       "DB_McpKeyboardSignals".sK5_GripperDrilledPart.sLedSWStatus := "DB_McpKeyboardSignals".sK5_GripperDrilledPart.sKeySWStatus;
       "DB_HmiKeyboardSignals".sK5a_GripperDrilledPartClose.sLedSWStatus := "DB_HmiKeyboardSignals".sK5a_GripperDrilledPartClose.sKeySWStatus;
       "DB_HmiKeyboardSignals".sK5b_GripperDrilledPartOpen.sLedSWStatus := "DB_HmiKeyboardSignals".sK5b_GripperDrilledPartOpen.sKeySWStatus;
   END_REGION

   REGION Undrilled Gripper        
       #sUndrilledGripper(iHoldPart := #sLoadGripperCloseReq,
                          iOpen := "DB_DigitalInputs".sLoadClampOpened.sSWStatus,
                          iCloseWithoutPart := "DB_DigitalInputs".sLoadClampNotClosedWithPart.sSWStatus,
                          iPulseTime := T#300ms,
                          iMonitorTime:=T#3s,
                          oClose => "DB_DigitalOutputs".sLoadClampClosing.sSWStatus,
                          oOpen => "DB_DigitalOutputs".sLoadClampOpening.sSWStatus,
                          oStateOpen => #sLoadOpen,
                          oStateClose => #sLoadClose,
                          oStateCloseWithPart => #sLoadCloseWithPart,
                          oErrorCode=>#sUndrilledGripperErrorCode);

       "LBP_AlarmMsgs".UserA[08].A70UUxx[14] := #sUndrilledGripperErrorCode = 1;    // Msg: 700814 "Loading Gripper Opening Timeout"
       "LBP_AlarmMsgs".UserA[08].A70UUxx[15] := #sUndrilledGripperErrorCode = 2;    // Msg: 700815 "Loading Gripper Closing Timeout"   
   END_REGION

   REGION Drilled Gripper
       #sDrilledGripper(iHoldPart := #sUnloadGripperCloseReq,
                        iOpen := "DB_DigitalInputs".sUnloadClampOpened.sSWStatus,
                        iCloseWithoutPart := "DB_DigitalInputs".sUnloadClampNotClosedWithPart.sSWStatus,
                        iPulseTime := T#300ms,
                        iMonitorTime:=T#3s,
                        oClose => "DB_DigitalOutputs".sUnloadClampClosing.sSWStatus,
                        oOpen => "DB_DigitalOutputs".sUnloadClampOpening.sSWStatus,
                        oStateOpen => #sUnLoadOpen,
                        oStateClose => #sUnLoadClose,
                        oStateCloseWithPart => #sUnLoadCloseWithPart,
                        oErrorCode=>#sDrilledGripperErrorCode);

       "LBP_AlarmMsgs".UserA[08].A70UUxx[16] := #sUndrilledGripperErrorCode = 1;    // Msg: 700816 "Unloading Gripper Opening Timeout"
       "LBP_AlarmMsgs".UserA[08].A70UUxx[17] := #sUndrilledGripperErrorCode = 2;    // Msg: 700817 "Unloading Gripper Closing Timeout"   
   END_REGION

   REGION Blowing
       // Blowing from ISO Code
       IF "LBP_Chan1".MDyn[96] THEN
           #sBlowingISO := TRUE;
       ELSIF "LBP_Chan1".MDyn[97] OR "LBP_Chan1".A_Reset THEN
           #sBlowingISO := FALSE;
       END_IF;

       #sRT_BlowingCmdHMI(CLK := "DB_HMICmd".BlowingCmd);

       #sBlowingTimerCmdHMI(IN := #sRT_BlowingCmdHMI.Q,
                      PT := REAL_TO_DINT("DB_HMISetting".BlowingSetpoint));

       "DB_DigitalOutputs".sBlowing.sSWStatus := "DB_LoaderShuttle1".oBlowingReq
       OR "DB_LoaderShuttle2".oBlowingReq
       OR "DB_LoaderFixture".oBlowingReq
       OR  #sBlowingTimerCmdHMI.Q;

       "DB_HMICmd".BlowingCmd := FALSE;
   END_REGION

   REGION Gripper Status
       IF "DB_LoaderShuttle1".sMain.oGripperAxisRequest AND #sGripperStatus.Available AND NOT "DB_CommPLC_ISO".sAxisReservedbyNC THEN
           #sGripperStatus.Available := FALSE;
           #sGripperStatus.DrivedByShuttle1 := TRUE;
           #sGripperStatus.DrivedByShuttle2 := FALSE;
           #sGripperStatus.DrivedByFixture := FALSE;
       ELSIF "DB_LoaderShuttle2".sMain.oGripperAxisRequest AND #sGripperStatus.Available  AND NOT "DB_CommPLC_ISO".sAxisReservedbyNC THEN
           #sGripperStatus.Available := FALSE;
           #sGripperStatus.DrivedByShuttle1 := FALSE;
           #sGripperStatus.DrivedByShuttle2 := TRUE;
           #sGripperStatus.DrivedByFixture := FALSE;
       ELSIF #sGripperReq.ByFixture AND #sGripperStatus.Available  AND "DB_CommPLC_ISO".sAxisReservedbyNC THEN
           #sGripperStatus.Available := FALSE;
           #sGripperStatus.DrivedByShuttle1 := FALSE;
           #sGripperStatus.DrivedByShuttle2 := FALSE;
           #sGripperStatus.DrivedByFixture := TRUE;
       END_IF;

       IF "DB_LoaderShuttle1".sMain.oGripperAxisRelease THEN
           #sGripperStatus.DrivedByShuttle1 := FALSE;
       END_IF;
       IF "DB_LoaderShuttle2".sMain.sGripperAxisRelease THEN
           #sGripperStatus.DrivedByShuttle2 := FALSE;
       END_IF;
       IF NOT #sGripperReq.ByFixture THEN
           #sGripperStatus.DrivedByFixture := FALSE;
       END_IF;

       IF NOT #sGripperStatus.DrivedByShuttle1
           AND NOT #sGripperStatus.DrivedByShuttle2
           AND NOT #sGripperStatus.DrivedByFixture THEN
           #sGripperStatus.Available := TRUE;
           #sGripperStatus.DrivedByShuttle1 := FALSE;
           #sGripperStatus.DrivedByShuttle2 := FALSE;
           #sGripperStatus.DrivedByFixture := FALSE;
       END_IF;
   END_REGION
END_FUNCTION_BLOCK

FUNCTION_BLOCK "FB_Gripper"   // FB54, SCL
{ S7_Optimized_Access := 'TRUE' }
// stored: MemoryReserve 100, SetENOAutomatically false
   VAR_INPUT
      iHoldPart : Bool;   // Hold Part Request
      iOpen : Bool;   // Shim Plate Opened (DI)
      iCloseWithoutPart : Bool;   // Shim Plate Closed with Part (DI)
      iPulseTime : Time;   // Pulse before Closing Time (WFA ???)
      iMonitorTime : Time;
   END_VAR
   VAR_OUTPUT
      oClose : Bool;   // Closing Request (DO)
      oOpen : Bool;   // Openeing Request (DO)
      oStateOpen : Bool;   // Opened Status
      oStateClose : Bool;   // Closed Status
      oStateCloseWithPart : Bool;   // Closed with Part Status
      oErrorCode { ExternalAccessible := 'False'; ExternalVisible := 'False'; ExternalWritable := 'False'} : Int;
   END_VAR
   VAR
      sPulseTimer : TP_TIME;   // Pulse before Closing Timer (WFA ???)
      sMonitorTimer : TON_TIME;
   END_VAR
BEGIN
   REGION Description header 
       //==================================================================================
       // POSALUX Swiss SA / (C) Copyright 2025
       //----------------------------------------------------------------------------------
       // Title: Initialization of axis
       // Comment/Function: FB_LoaderShimPlate
       // Author: Fabien WALDT
       // Engineering: TIA Portal v17
       //----------------------------------------------------------------------------------
       // Change log table:
       // Version  | Date     | Expert in charge | Changes applied
       // ---------|----------|------------------|-----------------------------------------
       // 00.00.01 | 20250423 | WFA              | First released version
       // =================================================================================
   END_REGION

   REGION Open - Close request
       // Close request
       #sPulseTimer(IN := #iHoldPart,
                   PT := #iPulseTime);
       #oClose := #sPulseTimer.Q AND #iHoldPart;

       // Open Request
       #oOpen := NOT #iHoldPart AND NOT #iOpen;
   END_REGION

   REGION Gripper States
       // State : Open
       #oStateOpen := #iOpen;

       //State : Close
       #oStateClose := NOT #iOpen AND NOT #oOpen AND NOT #oClose AND #iCloseWithoutPart ;

       // State : Close with Part
       #oStateCloseWithPart := NOT #iOpen AND NOT #oOpen AND NOT #oClose AND NOT #iCloseWithoutPart;
   END_REGION

   REGION Monitoring Timer
       #sMonitorTimer(IN := (#oOpen AND NOT #oStateOpen) OR
                      (#oClose AND (NOT #oStateClose AND NOT #oStateCloseWithPart) OR
                      (NOT #oStateOpen AND NOT #oStateClose AND NOT #oStateCloseWithPart) OR
                      (#oStateOpen AND (#oStateClose OR #oStateCloseWithPart))),
                      PT := #iMonitorTime);
   END_REGION

   REGION Error Codes
       #oErrorCode := 0;        // Code 0: No Error
       IF #oOpen AND #sMonitorTimer.Q THEN
           #oErrorCode := 1;    // Code 1: Error Open Command Plus
       ELSIF #oClose AND #sMonitorTimer.Q THEN
           #oErrorCode := 2;    // Code 2: Error Close Command Minus
       ELSIF NOT #oStateOpen AND NOT #oStateClose AND NOT #oStateCloseWithPart AND #sMonitorTimer.Q THEN
           #oErrorCode := 3;    // Code 3: Error Timeout Position OFF   
       ELSIF #oStateOpen AND (#oStateClose OR #oStateCloseWithPart) AND #sMonitorTimer.Q THEN
           #oErrorCode := 4;    // Code 4: Error Timeout Position ON       
       END_IF;
   END_REGION
END_FUNCTION_BLOCK

FUNCTION_BLOCK "FB_GestionFixture"   // FB49, SCL
{ S7_Optimized_Access := 'TRUE' }
// stored: MemoryReserve 100, SetENOAutomatically false
   VAR RETAIN
      sFixtureHold : Bool;
   END_VAR
   VAR
      sFixtureVacuum : Bool;
      sFixtureBlowing : Bool;
      sFixtureStandard { S7_SetPoint := 'True'} : "FB_Fixture";
      sFixtureStandardErrorCode { S7_SetPoint := 'True'} : Int;
      sFixturePartControl : "FB_PartPresenceCtrl";
      sRT_VacuumStartReq { S7_SetPoint := 'True'} : R_TRIG;
      sRT_VacuumStopReq { S7_SetPoint := 'True'} : R_TRIG;
   END_VAR
   VAR_TEMP
      tFixtureOpenAllowed : Bool;
      tFixtureCloseAllowed : Bool;
      tNull : Bool;
   END_VAR
   VAR CONSTANT
      B_AXIS_POSITION_MIN : Real := 0.0;   // B Axis Pos. Min to allow fixture opening
      B_AXIS_POSITION_MAX : Real := 15.0;   // B Axis Pos. Max to allow fixture opening
      V_AXIS_POSITION_MIN : Real := -1.0;   // V Axis Pos. Min to allow fixture opening/closing
      V_AXIS_POSITION_MAX : Real := 15.0;   // V Axis Pos. Max to allow fixture opening/closing
      W_AXIS_POSITION_MIN : Real := 0.0;   // W Axis Pos. Min to allow fixture opening/closing
      W_AXIS_POSITION_MAX : Real := 15.0;   // W Axis Pos. Max to allow fixture opening/closing
   END_VAR
BEGIN
   REGION Description header 
       //==================================================================================
       // POSALUX Swiss SA / (C) Copyright 2025
       //----------------------------------------------------------------------------------
       // Title: Structure sequence
       // Comment/Function: 
       //
       // Author: Fabien Waldt
       // Engineering: TIA Portal v17
       //----------------------------------------------------------------------------------
       // Change log table:
       // Version  | Date     | Expert in charge | Changes applied
       // ---------|----------|------------------|------------------------------------
       // 00.00.01 | 20250219 | WFA              | First released version
       // ==================================================================================
   END_REGION

   REGION
       #tFixtureOpenAllowed := ("DB_AxisPosition".sAxis04_B."$AA_IM" >= #B_AXIS_POSITION_MIN  AND "DB_AxisPosition".sAxis04_B."$AA_IM" <= #B_AXIS_POSITION_MAX)
                           AND ("DB_AxisPosition".sAxis07_V."$AA_IM" >= #V_AXIS_POSITION_MIN  AND "DB_AxisPosition".sAxis08_W."$AA_IM" >= #W_AXIS_POSITION_MIN);
       #tFixtureCloseAllowed := ("DB_AxisPosition".sAxis07_V."$AA_IM" >= #V_AXIS_POSITION_MIN AND "DB_AxisPosition".sAxis08_W."$AA_IM" >= #W_AXIS_POSITION_MIN);
   END_REGION

   REGION HOLD CLAMP
       REGION F_Hold Key Disable + channel switch Key[7]
       // Hold Key[7] disable 
           "DB_McpKeyboardSignals".sK7_FixtureClamp.sKeyDisable := "LBP_Chan1".E_ProgRunning OR "DB_GestionWorkingModes".sMCP_KxxKeysDisable;
            "DB_HmiKeyboardSignals".sK7_FixtureClamp.sKeyDisable := "LBP_Chan1".E_ProgRunning;
       // Force toggle Key[7] when hold is active    
            "DB_McpKeyboardSignals".sK7_FixtureClamp.sKeySWToggleStatus := #sFixtureHold;
            "DB_HmiKeyboardSignals".sK7_FixtureClamp.sKeySWToggleStatus := #sFixtureHold;
   END_REGION

   REGION Fixture 1 
       REGION Clamping Management
           // Hold signal for clamping - M84: Hold clamp
           IF #tFixtureCloseAllowed THEN
               IF "LBP_Chan1".MDyn[84]                                 // M84: Hold clamp
                   OR "DB_McpKeyboardSignals".sK7_FixtureClamp.sKeySWTogglePositiveFront
                   OR "DB_HmiKeyboardSignals".sK7_FixtureClamp.sKeySWTogglePositiveFront
                   OR "LBP_ModeGroup".A_REF
                   OR "DB_LoaderFixture".oFixtureCloseReq THEN
                   #sFixtureHold := TRUE;
                   "DB_McpKeyboardSignals".sK7_FixtureClamp.sKeySWToggleStatus := TRUE;
                   "DB_HmiKeyboardSignals".sK7_FixtureClamp.sKeySWToggleStatus := TRUE;
               END_IF;
           END_IF;
           // Release signal for clamping - M85: Release clamp
           IF #tFixtureOpenAllowed THEN
               IF "LBP_Chan1".MDyn[85]                                 // M85: Release clamp
                   OR "DB_McpKeyboardSignals".sK7_FixtureClamp.sKeySWToggleNegativeFront
                   OR "DB_HmiKeyboardSignals".sK7_FixtureClamp.sKeySWToggleNegativeFront
                   OR "DB_LoaderFixture".oFixtureOpenReq THEN
                   #sFixtureHold := FALSE;
                   "DB_McpKeyboardSignals".sK7_FixtureClamp.sKeySWToggleStatus := FALSE;
                   "DB_HmiKeyboardSignals".sK7_FixtureClamp.sKeySWToggleStatus := FALSE;
               END_IF;
           END_IF;
       END_REGION
   END_REGION
   END_REGION

   REGION F_Hold LED[7]
       "DB_McpKeyboardSignals".sK7_FixtureClamp.sLedSWStatus := #sFixtureHold;
       "DB_HmiKeyboardSignals".sK7_FixtureClamp.sLedSWStatus := #sFixtureHold;
   END_REGION

   REGION VACUUM
       REGION F_Vacuum Key Disable + Channel switch Key[8]
           // Vacuum Key[8] disable
           "DB_McpKeyboardSignals".sK8_FixtureVacuum.sKeyDisable := "LBP_Chan1".E_ProgRunning OR "DB_GestionWorkingModes".sMCP_KxxKeysDisable;
           "DB_HmiKeyboardSignals".sK8_FixtureVacuum.sKeyDisable := "LBP_Chan1".E_ProgRunning;

           // Force TOGGLE Key[8] when Vacuum is active    
           "DB_McpKeyboardSignals".sK8_FixtureVacuum.sKeySWToggleStatus := #sFixtureVacuum;
           "DB_HmiKeyboardSignals".sK8_FixtureVacuum.sKeySWToggleStatus := #sFixtureVacuum;
       END_REGION

       REGION Fixture 1
           #sRT_VacuumStartReq(CLK := "DB_LoaderFixture".sFixtureLoading.oVacuumStartReq);
           #sRT_VacuumStopReq(CLK := "DB_LoaderFixture".sFixtureUnloading.oVacuumStopReq);

           // Fixture Vacuum ON - M86: Vacuum ON
           IF "LBP_Chan1".MDyn[86]
               OR #sRT_VacuumStartReq.Q
               OR "DB_McpKeyboardSignals".sK8_FixtureVacuum.sKeySWTogglePositiveFront 
               OR "DB_HmiKeyboardSignals".sK8_FixtureVacuum.sKeySWTogglePositiveFront THEN
                   #sFixtureVacuum := TRUE;
                   "DB_McpKeyboardSignals".sK8_FixtureVacuum.sKeySWToggleStatus := TRUE;
                   "DB_HmiKeyboardSignals".sK8_FixtureVacuum.sKeySWToggleStatus := TRUE;
           END_IF;

           // Fixture Vacuum OFF (Station 1) - M87: Vacuum OFF
           IF "LBP_Chan1".MDyn[87]
               OR #sRT_VacuumStopReq.Q
               OR "DB_McpKeyboardSignals".sK8_FixtureVacuum.sKeySWToggleNegativeFront 
               OR "DB_HmiKeyboardSignals".sK8_FixtureVacuum.sKeySWToggleNegativeFront THEN
                   #sFixtureVacuum := FALSE;
                   "DB_McpKeyboardSignals".sK8_FixtureVacuum.sKeySWToggleStatus := FALSE;
                   "DB_HmiKeyboardSignals".sK8_FixtureVacuum.sKeySWToggleStatus := FALSE;
           END_IF;
       END_REGION

       REGION F_Vacuum LED[8]
           "DB_McpKeyboardSignals".sK8_FixtureVacuum.sLedSWStatus := #sFixtureVacuum;
           "DB_HmiKeyboardSignals".sK8_FixtureVacuum.sLedSWStatus := #sFixtureVacuum;
       END_REGION
   END_REGION

   REGION Standard Fixture
       #sFixtureStandard(iOpenCtrl := "DB_DigitalInputs".sClampingOpenCtrl.sSWStatus,
                         iCloseCtrl :="DB_DigitalOutputs".sClampingClosing.sSWStatus,
                         iHoldReq := #sFixtureHold,
                         iVacuumReq := #sFixtureVacuum,
                         iBlowingReq := #sFixtureBlowing,
                         iMonitorTime := T#2s,
                         oClampOpening => "DB_DigitalOutputs".sClampingOpening.sSWStatus,
                         oClampClosing => "DB_DigitalOutputs".sClampingClosing.sSWStatus,
                         oVacuumActivation => "DB_DigitalOutputs".sSuction.sSWStatus,
                         oBlowingActivation => #tNull, // No Blowing
                         oErrorCode => #sFixtureStandardErrorCode);
   END_REGION

   REGION Station 1 Fixture Alarms
       "LBP_AlarmMsgs".UserA[08].A70UUxx[12] := #sFixtureStandardErrorCode = 1;    // Msg: 700812 "Fixture Opening Timeout"
       "LBP_AlarmMsgs".UserA[08].A70UUxx[13] := #sFixtureStandardErrorCode = 2;    // Msg: 700813 "Fixture Closing Timeout"
   END_REGION

   REGION Fixture Part Control
       // Measure > iProdOK_LimHigh                          => Bad Positionning
       // iProdOK_LimLow <= Measure <= iProdOK_LimHigh       => Good part
       // NOT (iProdOK_LimLow <= Measure <= iProdOK_LimHigh) => Bad part
       // iProdMissing <= Measure <= iProdOK_LimLow          => Missing Backwall   (NOT POSSIBLE FOR FL.0153)
       // Measure < iProdMissing                             => Missing Part       (NOT POSSIBLE FOR FL.0153)
       // Teach-in :
           // ProdOK_LimHigh
           // ProdOK_LimLow
           // ProdMissing  (NOT USED FOR FL.0153)

       #sFixturePartControl.iProdOK_LimHigh := 25000; // WFA A supprimer quand recette OK
       #sFixturePartControl.iProdOK_LimLow := 9500; // WFA A supprimer quand recette OK
       // Voir dans FB_Recipe les transferts des limites High et Low

       #sFixturePartControl("iStart Control" := ("DB_LoaderFixture".oFixtureCloseReq OR "DB_DigitalOutputs".sClampingClosing.sSWStatus),             // M84: Hold clamp
                            iMeasureValue := "DB_AnalogInputs".sAxisB_ClampingPart.sSWRealValue,
                            iProdOK_LimHigh := #sFixturePartControl.iProdOK_LimHigh,
                            iProdOK_LimLow := #sFixturePartControl.iProdOK_LimLow,
                            iProdMissing:= #sFixturePartControl.iProdMissing,
                            oGoodPart => #sFixturePartControl.oGoodPart,
                            oBadpart => #sFixturePartControl.oBadpart);
   END_REGION

    REGION RID Fixture mvt
         "LBP_AlarmMsgs".Chan[1].RID[10] := #sFixtureStandard.oClampClosing AND NOT #sFixtureStandard.iCloseCtrl
         OR #sFixtureStandard.oClampOpening AND NOT #sFixtureStandard.iOpenCtrl;
    END_REGION
END_FUNCTION_BLOCK

FUNCTION_BLOCK "FB_Fixture"   // FB37, SCL
{ S7_Optimized_Access := 'TRUE' }
// stored: MemoryReserve 100, SetENOAutomatically false
   VAR_INPUT
      iOpenCtrl { ExternalAccessible := 'False'; ExternalVisible := 'False'; ExternalWritable := 'False'} : Bool;
      iCloseCtrl { ExternalAccessible := 'False'; ExternalVisible := 'False'; ExternalWritable := 'False'} : Bool;
      iHoldReq : Bool;   // Hold Request
      iVacuumReq : Bool;   // Vacuum Request
      iBlowingReq : Bool;   // Blowing Request
      iMonitorTime : Time;
   END_VAR
   VAR_OUTPUT
      oClampOpening : Bool;   // Clamp Opening
      oClampClosing : Bool;   // Clamp Closing
      oVacuumActivation : Bool;   // Vacuum Activation
      oBlowingActivation : Bool;   // Blowing Activation
      oErrorCode { ExternalAccessible := 'False'; ExternalVisible := 'False'; ExternalWritable := 'False'} : Int;
   END_VAR
   VAR
      sMonitorTimer : TON_TIME;
   END_VAR
BEGIN
   REGION Description header 
       //==================================================================================
       // POSALUX Swiss SA / (C) Copyright 2025
       //----------------------------------------------------------------------------------
       // Title: FB_Fixture
       // Comment/Function: 
       // Author: Fabien WALDT
       // Engineering: TIA Portal v17
       //----------------------------------------------------------------------------------
       // Change log table:
       // Version  | Date     | Expert in charge | Changes applied
       // ---------|----------|------------------|-----------------------------------------
       // 00.00.01 | 20250502 | WFA              | First released version
       // =================================================================================
   END_REGION

   REGION Init
   // Outputs Initialisation
   #oClampOpening := FALSE;
   #oClampClosing := FALSE;
   #oVacuumActivation := FALSE;
   #oBlowingActivation := FALSE;
   END_REGION

   REGION Clamp Opening - Closing
       IF #iHoldReq AND NOT "DB_MachineOptions".Fixture.Passive_Open THEN
           #oClampOpening := FALSE;
           #oClampClosing := TRUE;
       ELSIF NOT #iHoldReq AND NOT "DB_MachineOptions".Fixture.Passive_Open THEN
           #oClampOpening := TRUE;
           #oClampClosing := FALSE;
       END_IF;
   END_REGION

   REGION Vacuum Activation
       #oVacuumActivation := #iVacuumReq;
   END_REGION

   REGION Blowing Activation
       #oBlowingActivation := #iBlowingReq;
   END_REGION

   REGION Monitoring Timer
       #sMonitorTimer(IN := (#oClampOpening AND NOT #iOpenCtrl) 
                         OR (#oClampClosing AND NOT #iCloseCtrl)
                         OR (NOT #iOpenCtrl AND NOT #iCloseCtrl)
                         OR (#iOpenCtrl AND #iCloseCtrl),
                                PT := #iMonitorTime);
   END_REGION

   REGION Error Codes
       #oErrorCode := 0;        // Code 0: No Error
       IF #oClampOpening AND #sMonitorTimer.Q THEN
           #oErrorCode := 1;    // Code 1: Error Open Command Plus
       ELSIF #oClampClosing AND #sMonitorTimer.Q THEN
           #oErrorCode := 2;    // Code 2: Error Close Command Minus
       ELSIF NOT #iOpenCtrl AND NOT #iOpenCtrl AND #sMonitorTimer.Q THEN
           #oErrorCode := 3;    // Code 3: Error Timeout Position OFF   
       ELSIF #iOpenCtrl AND #iOpenCtrl AND #sMonitorTimer.Q THEN
           #oErrorCode := 4;    // Code 4: Error Timeout Position ON       
       END_IF;
   END_REGION
END_FUNCTION_BLOCK

FUNCTION_BLOCK "FB_PartPresenceCtrl"   // FB35, SCL
{ S7_Optimized_Access := 'TRUE' }
// stored: MemoryReserve 100, SetENOAutomatically false
   VAR_INPUT
      "iStart Control" : Bool;
      iMeasureValue : Real;
      iProdOK_LimHigh : Real;
      iProdOK_LimLow : Real;
      iProdMissing : Real;
   END_VAR
   VAR_OUTPUT
      oGoodPart : Bool;
      oBadpart : Bool;
   END_VAR
   VAR
      sRT_StartControl : R_TRIG;
      sBadPositioning { S7_SetPoint := 'True'} : Bool;
      sMissingBW { S7_SetPoint := 'True'} : Bool;
      sMissingPart : Bool;
      sStabilisationTime : TON_TIME;
   END_VAR
   VAR CONSTANT
      STABILISATION_TIME : Time := T#700ms;
   END_VAR
BEGIN
   REGION Description header 
       //==================================================================================
       // POSALUX Swiss SA / (C) Copyright 2025
       //----------------------------------------------------------------------------------
       // Title: CheckTimeout
       // Comment/Function: FB_PartPresenceCtrl
       //                   
       // Author: Fabien WALDT
       // Engineering: TIA Portal v19
       //----------------------------------------------------------------------------------
       // Change log table:
       // Version  | Date     | Expert in charge | Changes applied
       // ---------|----------|------------------|-----------------------------------------
       // 00.00.01 | 20250915 | WFA              | First released version
       // =================================================================================
   END_REGION

   REGION RT Start Cycle
       #sRT_StartControl(CLK := #"iStart Control");

      // IF #sRT_StartControl.Q THEN
       IF NOT #"iStart Control" THEN
           #oGoodPart := FALSE;
           #oBadpart := FALSE;
           #sBadPositioning := FALSE;
           #sMissingBW := FALSE;
           #sMissingPart := FALSE;
       END_IF;
   END_REGION

   REGION Stabilsation Time
       #sStabilisationTime(IN := #"iStart Control",
                           PT := #STABILISATION_TIME);
   END_REGION ;

   REGION Check Part
       IF #sStabilisationTime.Q THEN
           IF #iMeasureValue >= #iProdOK_LimLow AND #iMeasureValue <= #iProdOK_LimHigh THEN
               #oGoodPart := TRUE;
               #oBadpart := FALSE;
           ELSE
               #oGoodPart := FALSE;
               #oBadpart := TRUE;
               IF #iMeasureValue > #iProdOK_LimHigh THEN
                   #sBadPositioning := TRUE;
               ELSIF #iMeasureValue < #iProdMissing THEN
                   #sMissingPart := TRUE;
               ELSE
                   #sMissingBW := TRUE;
               END_IF;
           END_IF;
       END_IF;
   END_REGION
END_FUNCTION_BLOCK

FUNCTION_BLOCK "FB_TimeMeasure"   // FB51, SCL
{ S7_Optimized_Access := 'TRUE' }
// stored: AutoNumber false, MemoryReserve 100, SetENOAutomatically false
   VAR_INPUT
      iImpulsion : Bool;
      iPLC_DateAndTime : DTL;
   END_VAR
   VAR
      sRT_Impuls : R_TRIG;
      sRT_Impuls1 : R_TRIG;
      sRT_Impuls2 { S7_SetPoint := 'True'} : R_TRIG;
      sTime1 { S7_SetPoint := 'True'} : DTL;
      sTime2 : DTL;
      sDeltaTime : LTime;
      sToggleStatus : Bool;
   END_VAR
BEGIN
   REGION Description header 
       //==================================================================================
       // POSALUX Swiss SA / (C) Copyright 2026
       //----------------------------------------------------------------------------------
       // Title: FB_TimeMeasure
       // Comment/Function: This function allows:
       //                      - Counting Time between 2 pulses
       //
       // Author: Fabien Waldt
       // Engineering: TIA Portal v20
       //----------------------------------------------------------------------------------
       // Change log table:
       // Version  | Date     | Expert in charge | Changes applied
       // ---------|----------|------------------|------------------------------------
       // 00.00.01 | 20261211 | WFA              | First released version
       // ==================================================================================
   END_REGION

   REGION Delta time calculation
       // Rising edge detection
       #sRT_Impuls(CLK := #iImpulsion);

       // Toggle state update
       IF #sRT_Impuls.Q THEN
           #sToggleStatus := NOT #sToggleStatus;
       END_IF;
       #sRT_Impuls1(CLK := #sToggleStatus);
       #sRT_Impuls2(CLK := NOT #sToggleStatus);

       // Timestamp of the first rising edge
       IF #sRT_Impuls1.Q THEN
           #sTime1 := #iPLC_DateAndTime;
       END_IF;

       // Timestamp of the second rising edge + calculation
       IF #sRT_Impuls2.Q THEN
           #sTime2 := #iPLC_DateAndTime;
           #sDeltaTime := #sTime2 - #sTime1;
       END_IF;
   END_REGION
END_FUNCTION_BLOCK

FUNCTION_BLOCK "FB_LoaderFixtureMain"   // FB208, SCL
{ S7_Optimized_Access := 'TRUE' }
// stored: AutoNumber false, MemoryReserve 100, SetENOAutomatically false
   VAR
      sSynchroMode : Bool;
      sSynchroPosition : Bool;
      sTimeMeasure : "FB_TimeMeasure";
      sBlowingNotFinished { S7_SetPoint := 'True'} : Bool;
      sLoadingNotFinished : Bool;
      sUnloadingNotFinished : Bool;
      sReleaseNotFinished : Bool;
      sV_InitNotFinished : Bool;
      sW_InitNotFinished : Bool;
   END_VAR
BEGIN
   REGION Description header 
       //==================================================================================
       // POSALUX Swiss SA / (C) Copyright 2025
       //----------------------------------------------------------------------------------
       // Title: 
       // Comment/Function: 
       // Author: Fabien WALDT
       // Engineering: TIA Portal v17
       //----------------------------------------------------------------------------------
       // Change log table:
       // Version  | Date     | Expert in charge | Changes applied
       // ---------|----------|------------------|-----------------------------------------
       // 00.00.01 | 20251013 | WFA              | First released version
       // =================================================================================
   END_REGION

   REGION Options
       // Fixture
       "DB_LoaderOptions".Fixture.UnloadingDisabled := FALSE;
       "DB_LoaderOptions".Fixture.LoadingDisabled := FALSE;
       "DB_LoaderOptions".Fixture.BlowingDisabled := FALSE;
       "DB_LoaderOptions".Fixture.ReleaseDisabled := TRUE;
       "DB_LoaderOptions".Fixture.V_InitDisabled := FALSE;
       "DB_LoaderOptions".Fixture.W_InitDisabled := FALSE;
   END_REGION

   REGION History Activation
       // Fixture
       "DB_LoaderFixture".sFixtureUnloading.sHistory.Activation := TRUE;
       "DB_LoaderFixture".sFixtureLoading.sHistory.Activation := TRUE;
       "DB_LoaderFixture".sFixtureBlowing.sHistory.Activation := TRUE;
       "DB_LoaderFixture".sFixtureRelease.sHistory.Activation := TRUE;
       "DB_LoaderFixture".sFixtureV_Init.sHistory.Activation := TRUE;
       "DB_LoaderFixture".sFixtureW_Init.sHistory.Activation := TRUE;
   END_REGION

   REGION Fixture
       "DB_LoaderFixture"(iAxisV_Moving:="DB_LoaderAxis".sVPositioning,
                          iAxisV_InPos:="DB_LoaderAxis".sVInPos,
                          iAxisW_Moving:="DB_LoaderAxis".sWPositioning,
                          iAxisW_InPos:="DB_LoaderAxis".sWInPos,
                          oFixtureOpenReq=>"DB_LoaderFixture".oFixtureOpenReq,
                          oFixtureCloseReq=>"DB_LoaderFixture".oFixtureCloseReq,
                          oLoadGripperOpenReq=>"DB_LoaderFixture".oLoadGripperOpenReq,
                          oUnloadGripperCloseReq=>"DB_LoaderFixture".oUnloadGripperCloseReq,
                          oBlowingReq=>"DB_LoaderFixture".oBlowingReq,
                          oAxisV_StartReq=>"DB_LoaderFixture".oAxisV_StartReq,
                          oAxisV_PosSetPoint=>"DB_LoaderFixture".oAxisV_PosSetPoint,
                          oAxisW_StartReq=>"DB_LoaderFixture".oAxisW_StartReq,
                          oAxisW_PosSetPoint=>"DB_LoaderFixture".oAxisW_PosSetPoint);
   END_REGION

   REGION Sequences Not Finished
       IF "DB_LoaderFixture".sFixtureMain.sMemoBlowingRequest THEN
           #sBlowingNotFinished :=
           ("LBP_AlarmMsgs".UserA[08].A70UUxx[11]
           OR "LBP_AlarmMsgs".UserA[08].A70UUxx[10]
           OR "LBP_AlarmMsgs".UserA[08].A70UUxx[12]);
       END_IF;

       IF "DB_LoaderFixture".sFixtureMain.sMemoLoadingRequest THEN
           #sLoadingNotFinished :=
           ("LBP_AlarmMsgs".UserA[08].A70UUxx[11]
           OR "LBP_AlarmMsgs".UserA[08].A70UUxx[10]
           OR "LBP_AlarmMsgs".UserA[08].A70UUxx[12]
           OR "LBP_AlarmMsgs".UserA[08].A70UUxx[14]
           OR "LBP_AlarmMsgs".UserA[08].A70UUxx[13]);
           //  OR "LBP_AlarmMsgs".UserA[04].A70UUxx[26]
       END_IF;

       IF "DB_LoaderFixture".sFixtureMain.sMemoUnloadingRequest THEN
           #sUnloadingNotFinished := 
           ("LBP_AlarmMsgs".UserA[08].A70UUxx[11]
           OR "LBP_AlarmMsgs".UserA[08].A70UUxx[10]
           OR "LBP_AlarmMsgs".UserA[08].A70UUxx[12]
           OR "LBP_AlarmMsgs".UserA[08].A70UUxx[17]);
       END_IF;

       #sReleaseNotFinished := "DB_LoaderFixture".sFixtureRelease.sInterface.SequenceRun AND
       ("LBP_AlarmMsgs".UserA[08].A70UUxx[11]
       OR "LBP_AlarmMsgs".UserA[08].A70UUxx[10]);

       #sV_InitNotFinished := "DB_LoaderFixture".sFixtureV_Init.sInterface.SequenceRun AND
       ("LBP_AlarmMsgs".UserA[08].A70UUxx[10]);

       #sW_InitNotFinished := "DB_LoaderFixture".sFixtureW_Init.sInterface.SequenceRun AND
       ("LBP_AlarmMsgs".UserA[08].A70UUxx[11]);
   END_REGION

   REGION Alarm Not Ready
       // 700515 Gripper not ready for unloading
       IF "DB_LoaderFixture".sFixtureMain.sMemoUnloadingRequest AND NOT "DB_LoaderFixture".sFixtureMain.iGripperReadyForUnloading THEN
           "LBP_AlarmMsgs".UserA[05].A70UUxx[15] := TRUE;
       ELSE
           "LBP_AlarmMsgs".UserA[05].A70UUxx[15] := FALSE;
       END_IF;

       // 700516 Gripper not ready for loading
       IF "DB_LoaderFixture".sFixtureMain.sMemoLoadingRequest AND NOT "DB_LoaderFixture".sFixtureMain.iGripperReadyForLoading THEN
           "LBP_AlarmMsgs".UserA[05].A70UUxx[16] := TRUE;
       ELSE
           "LBP_AlarmMsgs".UserA[05].A70UUxx[16] := FALSE;
       END_IF;

       // 700517 Gripper not ready for blowing
       IF "DB_LoaderFixture".sFixtureMain.sMemoBlowingRequest AND NOT "DB_LoaderFixture".sFixtureMain.iGripperReadyForBlowing THEN
           "LBP_AlarmMsgs".UserA[05].A70UUxx[17] := TRUE;
       ELSE
           "LBP_AlarmMsgs".UserA[05].A70UUxx[17] := FALSE;
       END_IF;

       // 700518 Gripper not ready for V Axis Init
       IF "DB_LoaderFixture".sFixtureMain.sMemoV_InitRequest AND NOT "DB_LoaderFixture".sFixtureMain.iGripperReadyForV_Init THEN
           "LBP_AlarmMsgs".UserA[05].A70UUxx[18] := TRUE;
       ELSE
           "LBP_AlarmMsgs".UserA[05].A70UUxx[18] := FALSE;
       END_IF;

       // 700519 Gripper not ready for W Axis Init 
       IF "DB_LoaderFixture".sFixtureMain.sMemoW_InitRequest AND NOT "DB_LoaderFixture".sFixtureMain.iGripperReadyForW_Init THEN
           "LBP_AlarmMsgs".UserA[05].A70UUxx[19] := TRUE;
       ELSE
           "LBP_AlarmMsgs".UserA[05].A70UUxx[19] := FALSE;
       END_IF;

       // 700520 Fixture not ready for unloading
       IF "DB_LoaderFixture".sFixtureMain.sMemoUnloadingRequest AND NOT "DB_LoaderFixture".sFixtureMain.iFixtureReadyForUnloading THEN
           "LBP_AlarmMsgs".UserA[05].A70UUxx[20] := TRUE;
       ELSE
           "LBP_AlarmMsgs".UserA[05].A70UUxx[20] := FALSE;
       END_IF;

       // 700521 Fixture not ready for loading
       IF "DB_LoaderFixture".sFixtureMain.sMemoLoadingRequest AND NOT "DB_LoaderFixture".sFixtureMain.iFixtureReadyForLoading THEN
           "LBP_AlarmMsgs".UserA[05].A70UUxx[21] := TRUE;
       ELSE
           "LBP_AlarmMsgs".UserA[05].A70UUxx[21] := FALSE;
       END_IF;

       // 700522 Fixture not ready for blowing  
       IF "DB_LoaderFixture".sFixtureMain.sMemoBlowingRequest AND NOT "DB_LoaderFixture".sFixtureMain.iFixtureReadyForBlowing THEN
           "LBP_AlarmMsgs".UserA[05].A70UUxx[22] := TRUE;
       ELSE
           "LBP_AlarmMsgs".UserA[05].A70UUxx[22] := FALSE;
       END_IF;

       // 700523 Fixture not ready for V Axis Init
       IF "DB_LoaderFixture".sFixtureMain.sMemoV_InitRequest AND NOT "DB_LoaderFixture".sFixtureMain.iFixtureReadyForV_Init THEN
           "LBP_AlarmMsgs".UserA[05].A70UUxx[23] := TRUE;
       ELSE
           "LBP_AlarmMsgs".UserA[05].A70UUxx[23] := FALSE;
       END_IF;

       // 700524 Fixture not ready for W Axis Init 
       IF "DB_LoaderFixture".sFixtureMain.sMemoW_InitRequest AND NOT "DB_LoaderFixture".sFixtureMain.iFixtureReadyForW_Init THEN
           "LBP_AlarmMsgs".UserA[05].A70UUxx[24] := TRUE;
       ELSE
           "LBP_AlarmMsgs".UserA[05].A70UUxx[24] := FALSE;
       END_IF;

       // 700525 Axis position not ready for unloading
       IF "DB_LoaderFixture".sFixtureMain.sMemoUnloadingRequest AND NOT "DB_LoaderFixture".sFixtureMain.iAxisReadyForUnloading THEN
           "LBP_AlarmMsgs".UserA[05].A70UUxx[25] := TRUE;
       ELSE
           "LBP_AlarmMsgs".UserA[05].A70UUxx[25] := FALSE;
       END_IF;

       // 700526 Axis position not ready for loading
       IF "DB_LoaderFixture".sFixtureMain.sMemoLoadingRequest AND NOT "DB_LoaderFixture".sFixtureMain.iAxisReadyForLoading THEN
           "LBP_AlarmMsgs".UserA[05].A70UUxx[26] := TRUE;
       ELSE
           "LBP_AlarmMsgs".UserA[05].A70UUxx[26] := FALSE;
       END_IF;

       // 700527 Axis position not ready for blowing
       IF "DB_LoaderFixture".sFixtureMain.sMemoBlowingRequest AND NOT "DB_LoaderFixture".sFixtureMain.iAxisReadyForBlowing THEN
           "LBP_AlarmMsgs".UserA[05].A70UUxx[27] := TRUE;
       ELSE
           "LBP_AlarmMsgs".UserA[05].A70UUxx[27] := FALSE;
       END_IF;

       // 700528 Axis position not ready for V Axis Init
       IF "DB_LoaderFixture".sFixtureMain.sMemoV_InitRequest AND NOT "DB_LoaderFixture".sFixtureMain.iAxisReadyForV_Init THEN
           "LBP_AlarmMsgs".UserA[05].A70UUxx[28] := TRUE;
       ELSE
           "LBP_AlarmMsgs".UserA[05].A70UUxx[28] := FALSE;
       END_IF;

       // 700529 Axis position not ready for W Axis Init 
       IF "DB_LoaderFixture".sFixtureMain.sMemoW_InitRequest AND NOT "DB_LoaderFixture".sFixtureMain.iAxisReadyForW_Init THEN
           "LBP_AlarmMsgs".UserA[05].A70UUxx[29] := TRUE;
       ELSE
           "LBP_AlarmMsgs".UserA[05].A70UUxx[29] := FALSE;
       END_IF;
   END_REGION
END_FUNCTION_BLOCK

FUNCTION_BLOCK "FB_LoaderFixture"   // FB207, SCL
{ S7_Optimized_Access := 'TRUE' }
// stored: AutoNumber false, MemoryReserve 100, SetENOAutomatically false
   VAR_INPUT
      iAxisV_Moving : Bool;
      iAxisV_InPos : Bool;
      iAxisW_Moving : Bool;
      iAxisW_InPos : Bool;
   END_VAR
   VAR_OUTPUT
      oFixtureOpenReq : Bool;
      oFixtureCloseReq : Bool;
      oLoadGripperOpenReq : Bool;
      oUnloadGripperCloseReq : Bool;
      oBlowingReq : Bool;
      oAxisV_StartReq : Bool;
      oAxisV_PosSetPoint : Real;
      oAxisW_StartReq : Bool;
      oAxisW_PosSetPoint : Real;
   END_VAR
   VAR
      sFixtureMain : "FB_FixtureUnloadLoad";
      sFixtureUnloading { S7_SetPoint := 'True'} : "FB_FixtureUnloading";
      sFixtureLoading { S7_SetPoint := 'True'} : "FB_FixtureLoading";
      sFixtureBlowing { S7_SetPoint := 'True'} : "FB_FixtureBlowing";
      sFixtureRelease { S7_SetPoint := 'True'} : "FB_FixtureRelease";
      sFixtureV_Init { S7_SetPoint := 'True'} : "FB_FixtureV_Init";
      sFixtureW_Init { S7_SetPoint := 'True'} : "FB_FixtureW_Init";
      sAxisVSafePos { S7_SetPoint := 'True'} : LReal;
      sStepPauseSeq { S7_SetPoint := 'True'} : Bool;
   END_VAR
   VAR_TEMP
      tAxisV_Position : Struct
         FixtureLoad : Bool;
         FixtureUnload : Bool;
         FixtureBlowing : Bool;
         FixtureSafe : Bool;
         ShuttleSafe : Bool;
         Shuttle1Blowing : Bool;
      END_STRUCT;
      tAxisW_Position : Struct
         FixtureLoad : Bool;
         FixtureUnload : Bool;
         FixtureBlowing : Bool;
         FixtureSafe : Bool;
         Approach : Bool;
      END_STRUCT;
   END_VAR
BEGIN
   REGION Axis V Safe Position
       IF "DB_LoaderShuttle1".sShuttlePosInt THEN
           #sAxisVSafePos := "DB_AxisPosMachinePLC".Axis_V.Shuttle_1.LoadUnload;
       ELSIF "DB_LoaderShuttle2".sShuttlePosInt THEN
           #sAxisVSafePos := "DB_AxisPosMachinePLC".Axis_V.Shuttle_2.LoadUnload;
       ELSE
           #sAxisVSafePos := "DB_AxisPosMachinePLC".Axis_V.Fixture.Safe;
       END_IF;
       // WFA revoir la gestion du Setpoint Safe en foncton de la shuttle
       #sAxisVSafePos := "DB_AxisPosMachinePLC".Axis_V.Fixture.Safe;
   END_REGION

   REGION Position Check
       REGION Axis V
           // Position : Fixture Load
           "FC_PositionCheck"(iAxisCurrentPos := "DB_AxisPosition".sAxis07_V."$AA_IM",
                              iAxisTargetPos := "DB_AxisPosMachinePLC".Axis_V.Fixture.Load,
                              iTolMin := 0.001,
                              iTolMax := 0.001,
                              iInPos => #tAxisV_Position.FixtureLoad);

           // Position : Fixture Unload
           "FC_PositionCheck"(iAxisCurrentPos := "DB_AxisPosition".sAxis07_V."$AA_IM",
                              iAxisTargetPos := "DB_AxisPosMachinePLC".Axis_V.Fixture.Unload,
                              iTolMin := 0.001,
                              iTolMax := 0.001,
                              iInPos => #tAxisV_Position.FixtureUnload);

           // Position : Fixture Blowing
           "FC_PositionCheck"(iAxisCurrentPos := "DB_AxisPosition".sAxis07_V."$AA_IM",
                              iAxisTargetPos := "DB_AxisPosMachinePLC".Axis_V.Fixture.Blowing,
                              iTolMin := 0.001,
                              iTolMax := 0.001,
                              iInPos => #tAxisV_Position.FixtureBlowing);

           // Position : Fixture Safe
           "FC_PositionCheck"(iAxisCurrentPos := "DB_AxisPosition".sAxis07_V."$AA_IM",
                              iAxisTargetPos := #sAxisVSafePos,
                              iTolMin := 0.001,
                              iTolMax := 0.001,
                              iInPos => #tAxisV_Position.FixtureSafe);

           // Position : Safe (Shuttle)
           "FC_PositionCheck"(iAxisCurrentPos := "DB_AxisPosition".sAxis07_V."$AA_IM",
                              iAxisTargetPos := "DB_AxisPosMachinePLC".Axis_V.Safe,
                              iTolMin := 0.001,
                              iTolMax := 0.001,
                              iInPos => #tAxisV_Position.ShuttleSafe);

           // Position : Blowing Shuttle 1
           "FC_PositionCheck"(iAxisCurrentPos := "DB_AxisPosition".sAxis07_V."$AA_IM",
                              iAxisTargetPos := "DB_AxisPosMachinePLC".Axis_V.Shuttle_1.Blowing,
                              iTolMin := 0.001,
                              iTolMax := 0.001,
                              iInPos => #tAxisV_Position.Shuttle1Blowing);
       END_REGION

       REGION Axis W
           // Position : Fixture Load
           "FC_PositionCheck"(iAxisCurrentPos := "DB_AxisPosition".sAxis08_W."$AA_IM",
                              iAxisTargetPos := "DB_AxisPosMachinePLC".Axis_W.Fixture.Load,
                              iTolMin := 0.001,
                              iTolMax := 0.001,
                              iInPos => #tAxisW_Position.FixtureLoad);

           // Position : Fixture Unload
           "FC_PositionCheck"(iAxisCurrentPos := "DB_AxisPosition".sAxis08_W."$AA_IM",
                              iAxisTargetPos := "DB_AxisPosMachinePLC".Axis_W.Fixture.Unload,
                              iTolMin := 0.001,
                              iTolMax := 0.001,
                              iInPos => #tAxisW_Position.FixtureUnload);

           // Position : Fixture Blowing
           "FC_PositionCheck"(iAxisCurrentPos := "DB_AxisPosition".sAxis08_W."$AA_IM",
                              iAxisTargetPos := "DB_AxisPosMachinePLC".Axis_W.Fixture.Blowing,
                              iTolMin := 0.001,
                              iTolMax := 0.001,
                              iInPos => #tAxisW_Position.FixtureBlowing);

           // Position : Fixture Safe
           "FC_PositionCheck"(iAxisCurrentPos := "DB_AxisPosition".sAxis08_W."$AA_IM",
                              iAxisTargetPos := "DB_AxisPosMachinePLC".Axis_W.Fixture.Safe,
                              iTolMin := 0.001,
                              iTolMax := 0.001,
                              iInPos => #tAxisW_Position.FixtureSafe);

           // Position : Approach (confondu avec load/unload)
           "FC_PositionCheck"(iAxisCurrentPos := "DB_AxisPosition".sAxis08_W."$AA_IM",
                              iAxisTargetPos := "DB_AxisPosMachinePLC".Axis_W.Fixture.Approach,
                              iTolMin := 0.001,
                              iTolMax := 0.001,
                              iInPos => #tAxisW_Position.Approach);
       END_REGION
   END_REGION

   REGION Step Pause Sequence
       #sStepPauseSeq := "LBP_ModeGroup".E_JOG OR "DB_ExtraMissingPart".sGlobalExtraMissing;

       #sFixtureUnloading.iStepPause := #sStepPauseSeq;
       #sFixtureLoading.iStepPause := #sStepPauseSeq;
       #sFixtureBlowing.iStepPause := #sStepPauseSeq;
       #sFixtureRelease.iStepPause := #sStepPauseSeq;
       #sFixtureV_Init.iStepPause := #sStepPauseSeq;
       #sFixtureW_Init.iStepPause := #sStepPauseSeq;
   END_REGION

   REGION Fixture Unload Load
       // M33 : Fixture Unloading Request
       #sFixtureMain.iFixtureUnloadingRequest := "LBP_Chan1".MDyn[33];

       // M35 : Fixture Blowing Request
       #sFixtureMain.iFixtureBlowingRequest := "LBP_Chan1".MDyn[35];

       // M34 : Fixture Loading Request
       #sFixtureMain.iFixtureLoadingRequest := "LBP_Chan1".MDyn[34];

       // Release request (Release not used)
       #sFixtureMain.iFixtureReleaseRequest := FALSE;

       // M31 : Fixture V Init Request
       #sFixtureMain.iFixtureV_InitRequest := "LBP_Chan1".MDyn[31];

       // M32 : Fixture W Init Request
       #sFixtureMain.iFixtureW_InitRequest := "LBP_Chan1".MDyn[32];

       // Gripper ready for unloading
       #sFixtureMain.iGripperReadyForUnloading := ("DB_GestionGripper".sGripperStatus.Available OR "DB_GestionGripper".sGripperStatus.DrivedByFixture)
       AND ((NOT "DB_PartManagement".sPosition.sGripper.Drilled.Presence.Part AND NOT "DB_PartManagement".sPosition.sGripper.Drilled.Presence.BW AND "DB_GestionGripper".sDrilledGripper.oStateOpen AND "DB_WorkingModes".sEmptying)
       OR (NOT "DB_PartManagement".sPosition.sGripper.Drilled.Presence.Part AND NOT "DB_PartManagement".sPosition.sGripper.Drilled.Presence.BW AND "DB_PartManagement".sPosition.sGripper.Undrilled.Presence.Part AND "DB_PartManagement".sPosition.sGripper.Undrilled.Presence.BW AND "DB_GestionGripper".sDrilledGripper.oStateOpen AND "DB_WorkingModes".sNormal));

       // Gripper ready for loading
       #sFixtureMain.iGripperReadyForLoading := ("DB_GestionGripper".sGripperStatus.Available OR "DB_GestionGripper".sGripperStatus.DrivedByFixture)
       AND (("DB_PartManagement".sPosition.sGripper.Undrilled.Presence.Part AND "DB_PartManagement".sPosition.sGripper.Undrilled.Presence.BW AND "DB_WorkingModes".sFilling)
       OR ("DB_PartManagement".sPosition.sGripper.Undrilled.Presence.Part AND "DB_PartManagement".sPosition.sGripper.Undrilled.Presence.BW  AND ("DB_WorkingModes".sNormal OR "DB_WorkingModes".sEmptying)));

       // Gripper ready for blowing
       #sFixtureMain.iGripperReadyForBlowing := ("DB_GestionGripper".sGripperStatus.Available OR "DB_GestionGripper".sGripperStatus.DrivedByFixture)
       AND #sFixtureMain.iGripperReadyForLoading;

       // Gripper ready for Release (Release not used)
       #sFixtureMain.iGripperReadyForRelease := ("DB_GestionGripper".sGripperStatus.Available OR "DB_GestionGripper".sGripperStatus.DrivedByFixture);

       // Gripper ready for V Init
       #sFixtureMain.iGripperReadyForV_Init := ("DB_GestionGripper".sGripperStatus.Available OR "DB_GestionGripper".sGripperStatus.DrivedByFixture);

       // Gripper ready for W Init
       #sFixtureMain.iGripperReadyForW_Init := ("DB_GestionGripper".sGripperStatus.Available OR "DB_GestionGripper".sGripperStatus.DrivedByFixture);


       // Fixture ready for unloading
       #sFixtureMain.iFixtureReadyForUnloading := TRUE;

       // Fixture ready for loading
       #sFixtureMain.iFixtureReadyForLoading := "DB_PartManagement".sPosition.sFixtureEmpty;

       // Fixture ready for blowing
       #sFixtureMain.iFixtureReadyForBlowing := TRUE;

       // Fixture ready for Release (Release not used)
       #sFixtureMain.iFixtureReadyForRelease := TRUE;

       // Fixture ready for V Init
       #sFixtureMain.iFixtureReadyForV_Init := TRUE;

       // Fixture ready for W Init
       #sFixtureMain.iFixtureReadyForW_Init := TRUE;


       // Axis ready for Unloading
       #sFixtureMain.iAxisReadyForUnloading :=
       ("DB_AxisPosition".sAxis01_X."$AA_IM" = "DB_AxisPosMachineNC".Axis_X.Unload
       AND "DB_AxisPosition".sAxis02_Y."$AA_IM" = "DB_AxisPosMachineNC".Axis_Y.Unload
       AND "DB_AxisPosition".sAxis04_B."$AA_IM" = "DB_AxisPosMachineNC".Axis_B.Unload
       AND "DB_AxisPosition".sAxis03_ZM."$AA_IM" = "DB_AxisPosition".sAxis03_ZM."$MA_POS_LIMIT_MINUS2" + 1);

       // Axis ready for Loading
       #sFixtureMain.iAxisReadyForLoading :=
       ("DB_AxisPosition".sAxis01_X."$AA_IM" = "DB_AxisPosMachineNC".Axis_X.Load
       AND "DB_AxisPosition".sAxis02_Y."$AA_IM" = "DB_AxisPosMachineNC".Axis_Y.Load
       AND "DB_AxisPosition".sAxis04_B."$AA_IM" = "DB_AxisPosMachineNC".Axis_B.Load
       AND "DB_AxisPosition".sAxis03_ZM."$AA_IM" = "DB_AxisPosition".sAxis03_ZM."$MA_POS_LIMIT_MINUS2" + 1);

       // Axis ready for Blowing
       #sFixtureMain.iAxisReadyForBlowing :=
       ("DB_AxisPosition".sAxis01_X."$AA_IM" = "DB_AxisPosMachineNC".Axis_X.Blowing
       AND "DB_AxisPosition".sAxis02_Y."$AA_IM" = "DB_AxisPosMachineNC".Axis_Y.Blowing
       AND "DB_AxisPosition".sAxis04_B."$AA_IM" = "DB_AxisPosMachineNC".Axis_B.Blowing
       AND "DB_AxisPosition".sAxis03_ZM."$AA_IM" = "DB_AxisPosition".sAxis03_ZM."$MA_POS_LIMIT_MINUS2" + 1);

       // Axis ready for Release (Release not used)
       #sFixtureMain.iAxisReadyForRelease :=
       ("DB_AxisPosition".sAxis03_ZM."$AA_IM" = "DB_AxisPosition".sAxis03_ZM."$MA_POS_LIMIT_MINUS2" + 1
       AND "DB_AxisPosition".sAxis09_ZL."$AA_IM" = "DB_AxisPosMachineNC".Axis_ZL.Safe);

       // Axis ready for V Init
       #sFixtureMain.iAxisReadyForV_Init := TRUE;

       // Axis ready for W Init
       #sFixtureMain.iAxisReadyForW_Init := TRUE;

       #sFixtureMain(iFixtureUnloadingRequest:=#sFixtureMain.iFixtureUnloadingRequest,
                     iFixtureLoadingRequest:=#sFixtureMain.iFixtureLoadingRequest,
                     iFixtureBlowingRequest:=#sFixtureMain.iFixtureBlowingRequest,
                     iFixtureReleaseRequest:=#sFixtureMain.iFixtureReleaseRequest,
                     iFixtureV_InitRequest:=#sFixtureMain.iFixtureV_InitRequest,
                     iFixtureW_InitRequest:=#sFixtureMain.iFixtureW_InitRequest,
                     iWorkingModeFilling:="DB_WorkingModes".sFilling,
                     iWorkingModeEmptying:="DB_WorkingModes".sEmptying,
                     iGripperReadyForUnloading:=#sFixtureMain.iGripperReadyForUnloading,
                     iGripperReadyForLoading:=#sFixtureMain.iGripperReadyForLoading,
                     iGripperReadyForBlowing:=#sFixtureMain.iGripperReadyForBlowing,
                     iGripperReadyForRelease:=#sFixtureMain.iGripperReadyForRelease,
                     iGripperReadyForV_Init:=#sFixtureMain.iGripperReadyForV_Init,
                     iGripperReadyForW_Init:=#sFixtureMain.iGripperReadyForW_Init,
                     iFixtureReadyForUnloading:=#sFixtureMain.iFixtureReadyForUnloading,
                     iFixtureReadyForLoading:=#sFixtureMain.iFixtureReadyForLoading,
                     iFixtureReadyForBlowing:=#sFixtureMain.iFixtureReadyForBlowing,
                     iFixtureReadyForRelease:=#sFixtureMain.iFixtureReadyForRelease,
                     iFixtureReadyForV_Init:=#sFixtureMain.iFixtureReadyForV_Init,
                     iFixtureReadyForW_Init:=#sFixtureMain.iFixtureReadyForW_Init,
                     iAxisReadyForUnloading:=#sFixtureMain.iAxisReadyForUnloading,
                     iAxisReadyForLoading:=#sFixtureMain.iAxisReadyForLoading,
                     iAxisReadyForBlowing:=#sFixtureMain.iAxisReadyForBlowing,
                     iAxisReadyForRelease:=#sFixtureMain.iAxisReadyForRelease,
                     iAxisReadyForV_Init:=#sFixtureMain.iAxisReadyForV_Init,
                     iAxisReadyForW_Init:=#sFixtureMain.iAxisReadyForW_Init,
                     iAxisV_W_Available:="DB_GestionGripper".sGripperStatus.Available,
                     oAxisV_W_Reservation=>"DB_GestionGripper".sGripperReq.ByFixture,
                     oNC_RID1=>"LBP_AlarmMsgs".Chan[1].RID[8],
                     oNC_RID2=>"LBP_AlarmMsgs".Chan[1].RID[9],
                     ioFixtureUnloadingSeq:=#sFixtureUnloading.sInterface,
                     ioFixtureLoadingSeq:=#sFixtureLoading.sInterface,
                     ioFixtureBlowingSeq:=#sFixtureBlowing.sInterface,
                     ioFixtureReleaseSeq:=#sFixtureRelease.sInterface,
                     ioFixtureV_InitSeq:=#sFixtureV_Init.sInterface,
                     ioFixtureW_InitSeq:=#sFixtureW_Init.sInterface);
   END_REGION

   REGION Fixture Unloading
       // Unload Gripper Closed according to dry run working mode
        #sFixtureUnloading.iUnloadGripperClosed := ("DB_GestionGripper".sDrilledGripper.oStateCloseWithPart AND NOT "DB_WorkingModes".sDryRun)
        OR ("DB_GestionGripper".sDrilledGripper.oStateClose AND "DB_WorkingModes".sDryRun);

       #sFixtureUnloading(iStartSeqCond:= "DB_PowerOn".sMachineReadySoft AND NOT "DB_LoaderFixtureMain".sUnloadingNotFinished AND NOT "MCP1_In".reset,
                          iJobReq:=#sFixtureUnloading.sInterface.StartRequest,
                          iFixtureOpened:="DB_DigitalInputs".sClampingOpenCtrl.sSWStatus,
                          iUnloadGripperClosed:=#sFixtureUnloading.iUnloadGripperClosed, // WAF CHECK
                          iAxisV_FixtUnloadPos:=#tAxisV_Position.FixtureUnload,
                          iAxisV_FixtUnloadPosSetPoint:="DB_AxisPosMachinePLC".Axis_V.Fixture.Unload,
                          iAxisW_FixtSafePos:=#tAxisW_Position.FixtureSafe,
                          iAxisW_FixtSafePosSetPoint:="DB_AxisPosMachinePLC".Axis_W.Fixture.Safe,
                          iAxisW_FixtUnloadPos:=#tAxisW_Position.FixtureUnload,
                          iAxisW_FixtUnloadPosSetPoint:="DB_AxisPosMachinePLC".Axis_W.Fixture.Unload,
                          iAxisV_Moving:=#iAxisV_Moving,
                          iAxisV_InPos:=#iAxisV_InPos,
                          iAxisW_Moving:=#iAxisW_Moving,
                          iAxisW_InPos:=#iAxisW_InPos,
                          iPLC_DateAndTime:="DB_ReadDateAndTime".sDateAndTime,
                          iStepPause:=#sFixtureUnloading.iStepPause,
                          oFixtureOpenReq=>#sFixtureUnloading.oFixtureOpenReq,
                          oUnloadGripperCloseReq=>#sFixtureUnloading.oUnloadGripperCloseReq,
                          oVacuumStopReq=>#sFixtureUnloading.oVacuumStopReq,
                          oAxisV_StartReq=>#sFixtureUnloading.oAxisV_StartReq,
                          oAxisV_PosSetPoint=>#sFixtureUnloading.oAxisV_PosSetPoint,
                          oAxisW_StartReq=>#sFixtureUnloading.oAxisW_StartReq,
                          oAxisW_PosSetPoint=>#sFixtureUnloading.oAxisW_PosSetPoint);
   END_REGION

   REGION Fixture Loading
       // Load Gripper Closed according to dry run working mode
       #sFixtureLoading.iFixtureClosed := ("DB_GestionFixture".sFixturePartControl.oGoodPart AND NOT "DB_WorkingModes".sDryRun)
       OR ("DB_DigitalOutputs".sClampingClosing.sSWStatus AND ("DB_WorkingModes".sDryRun));

       #sFixtureLoading(iStartSeqCond := "DB_PowerOn".sMachineReadySoft AND NOT "DB_LoaderFixtureMain".sLoadingNotFinished AND NOT "MCP1_In".reset,
                        iJobReq := #sFixtureLoading.sInterface.StartRequest,
                        iFixtureOpened := "DB_DigitalInputs".sClampingOpenCtrl.sSWStatus,
                        iFixtureClosed := #sFixtureLoading.iFixtureClosed,
                        iLoadGripperOpened := "DB_GestionGripper".sUndrilledGripper.oStateOpen,
                        iAxisV_FixtLoadPos := #tAxisV_Position.FixtureLoad,
                        iAxisV_FixtLoadPosSetPoint := "DB_AxisPosMachinePLC".Axis_V.Fixture.Load,
                        iAxisW_FixtSafePos := #tAxisW_Position.FixtureSafe,
                        iAxisW_FixtSafePosSetPoint := "DB_AxisPosMachinePLC".Axis_W.Fixture.Safe,
                        iAxisW_FixtLoadPos := #tAxisW_Position.FixtureLoad,
                        iAxisW_FixtLoadPosSetPoint := "DB_AxisPosMachinePLC".Axis_W.Fixture.Load,
                        iAxisW_FixtApproachPos:=#tAxisW_Position.Approach,
                        iAxisW_FixtApproachPosSetPoint:="DB_AxisPosMachinePLC".Axis_W.Fixture.Approach,
                        iAxisV_Moving := #iAxisV_Moving,
                        iAxisV_InPos := #iAxisV_InPos,
                        iAxisW_Moving := #iAxisW_Moving,
                        iAxisW_InPos := #iAxisW_InPos,
                        iPLC_DateAndTime := "DB_ReadDateAndTime".sDateAndTime,
                        iStepPause := #sFixtureLoading.iStepPause,
                        oFixtureOpenReq => #sFixtureLoading.oFixtureOpenReq,
                        oFixtureCloseReq => #sFixtureLoading.oFixtureCloseReq,
                        oLoadGripperOpenReq => #sFixtureLoading.oLoadGripperOpenReq,
                        oVacuumStartReq=>#sFixtureLoading.oVacuumStartReq,
                        oAxisV_StartReq => #sFixtureLoading.oAxisV_StartReq,
                        oAxisV_PosSetPoint => #sFixtureLoading.oAxisV_PosSetPoint,
                        oAxisW_StartReq => #sFixtureLoading.oAxisW_StartReq,
                        oAxisW_PosSetPoint => #sFixtureLoading.oAxisW_PosSetPoint);
   END_REGION

   REGION Fixture Blowing
       #sFixtureBlowing(iStartSeqCond:= "DB_PowerOn".sMachineReadySoft AND NOT "DB_LoaderFixtureMain".sBlowingNotFinished AND NOT "MCP1_In".reset,
                        iJobReq:=#sFixtureBlowing.sInterface.StartRequest,
                        iFixtureOpened:="DB_DigitalInputs".sClampingOpenCtrl.sSWStatus,
                        iAxisV_FixtBlowingPos:=#tAxisV_Position.FixtureBlowing,
                        iAxisV_FixtBlowingPosSetPoint:="DB_AxisPosMachinePLC".Axis_V.Fixture.Blowing,
                        iAxisW_FixtSafePos:=#tAxisW_Position.FixtureSafe,
                        iAxisW_FixtSafePosSetPoint:="DB_AxisPosMachinePLC".Axis_W.Fixture.Safe,
                        iAxisW_FixtBlowPos:=#tAxisW_Position.FixtureBlowing,
                        iAxisW_FixtBlowPosSetPoint:="DB_AxisPosMachinePLC".Axis_W.Fixture.Blowing,
                        iAxisV_Moving:=#iAxisV_Moving,
                        iAxisV_InPos:=#iAxisV_InPos,
                        iAxisW_Moving:=#iAxisW_Moving,
                        iAxisW_InPos:=#iAxisW_InPos,
                        iBlowingTime:= DINT_TO_TIME(REAL_TO_DINT("DB_HMISetting".BlowingSetpoint)),
                        iPLC_DateAndTime:="DB_ReadDateAndTime".sDateAndTime,
                        iStepPause:=#sFixtureBlowing.iStepPause,
                        oFixtureOpenReq=>#sFixtureBlowing.oFixtureOpenReq,
                        oAxisV_StartReq=>#sFixtureBlowing.oAxisV_StartReq,
                        oAxisV_PosSetPoint=>#sFixtureBlowing.oAxisV_PosSetPoint,
                        oAxisW_StartReq=>#sFixtureBlowing.oAxisW_StartReq,
                        oAxisW_PosSetPoint=>#sFixtureBlowing.oAxisW_PosSetPoint,
                        oBlowingReq=>#sFixtureBlowing.oBlowingReq);
   END_REGION

   REGION Fixture Release  (Release not used)
       // Repli en position
       //  - Shuttle 1 (Pos. blowing Shuttle 1)
       //  - Shuttle 2 ( Pos Safe)
       IF "DB_LoaderShuttle1".sMain.sCurrent_Step_NB = 70 THEN
           #sFixtureRelease.iAxisV_SafePos := #tAxisV_Position.Shuttle1Blowing;
           #sFixtureRelease.iAxisV_SafePosSetPoint := "DB_AxisPosMachinePLC".Axis_V.Shuttle_1.Blowing;
       ELSE
           #sFixtureRelease.iAxisV_SafePos := #tAxisV_Position.ShuttleSafe;
           #sFixtureRelease.iAxisV_SafePosSetPoint := "DB_AxisPosMachinePLC".Axis_V.Safe;
       END_IF;

       #sFixtureRelease(iStartSeqCond := "DB_PowerOn".sMachineReadySoft AND NOT "DB_LoaderFixtureMain".sReleaseNotFinished AND NOT "MCP1_In".reset, // WAF TBD
                        iJobReq := #sFixtureRelease.sInterface.StartRequest,
                        iAxisV_SafePos := #sFixtureRelease.iAxisV_SafePos, // #tAxis_V_Position.Shuttle1Blowing, // #tAxis_V_Position.ShuttleSafe,
                        iAxisV_SafePosSetPoint := #sFixtureRelease.iAxisV_SafePosSetPoint, // "DB_AxisPosMachinePLC".Axis_V.Shuttle_1.Blowing,     // "DB_AxisPosMachinePLC".Axis_V.Safe,
                        iAxisW_FixtSafePos := #tAxisW_Position.FixtureSafe,
                        iAxisW_FixtSafePosSetPoint := "DB_AxisPosMachinePLC".Axis_W.Fixture.Safe,
                        iAxisV_Moving := #iAxisV_Moving,
                        iAxisV_InPos := #iAxisV_InPos,
                        iAxisW_Moving := #iAxisW_Moving,
                        iAxisW_InPos := #iAxisW_InPos,
                        iPLC_DateAndTime := "DB_ReadDateAndTime".sDateAndTime,
                        iStepPause := #sFixtureRelease.iStepPause,
                        oAxisV_StartReq => #sFixtureRelease.oAxisV_StartReq,
                        oAxisV_PosSetPoint => #sFixtureRelease.oAxisV_PosSetPoint,
                        oAxisW_StartReq => #sFixtureRelease.oAxisW_StartReq,
                        oAxisW_PosSetPoint => #sFixtureRelease.oAxisW_PosSetPoint);
   END_REGION

   REGION Fixture V Init
       #sFixtureV_Init(iStartSeqCond := "DB_PowerOn".sMachineReadySoft AND NOT "DB_LoaderFixtureMain".sV_InitNotFinished AND NOT "MCP1_In".reset,
                       iJobReq := #sFixtureV_Init.sInterface.StartRequest,
                       iAxisV_FixtSafePos := #tAxisV_Position.FixtureSafe,
                       iAxisV_FixtSafePosSetPoint := #sAxisVSafePos,
                       iAxisV_Moving := #iAxisV_Moving,
                       iAxisV_InPos := #iAxisV_InPos,
                       iPLC_DateAndTime := "DB_ReadDateAndTime".sDateAndTime,
                       iStepPause := #sFixtureV_Init.iStepPause,
                       oAxisV_StartReq => #sFixtureV_Init.oAxisV_StartReq,
                       oAxisV_PosSetPoint => #sFixtureV_Init.oAxisV_PosSetPoint);
   END_REGION

   REGION Fixture W Init
       #sFixtureW_Init(iStartSeqCond := "DB_PowerOn".sMachineReadySoft AND NOT "DB_LoaderFixtureMain".sW_InitNotFinished AND NOT "MCP1_In".reset,
                       iJobReq := #sFixtureW_Init.sInterface.StartRequest,
                       iAxisW_FixtSafePos := #tAxisW_Position.FixtureSafe,
                       iAxisW_FixtSafePosSetPoint := "DB_AxisPosMachinePLC".Axis_W.Fixture.Safe,
                       iAxisW_Moving := #iAxisW_Moving,
                       iAxisW_InPos := #iAxisW_InPos,
                       iPLC_DateAndTime := "DB_ReadDateAndTime".sDateAndTime,
                       iStepPause := #sFixtureW_Init.iStepPause,
                       iAxisW_StartReq => #sFixtureW_Init.iAxisW_StartReq,
                       iAxisW_PosSetPoint => #sFixtureW_Init.iAxisW_PosSetPoint);
   END_REGION

   REGION Axis U-V-W Start Request  
       // Axis V - Start Request
       #oAxisV_StartReq :=
       #sFixtureUnloading.oAxisV_StartReq
       OR #sFixtureLoading.oAxisV_StartReq
       OR #sFixtureBlowing.oAxisV_StartReq
       OR #sFixtureRelease.oAxisV_StartReq
       OR #sFixtureV_Init.oAxisV_StartReq;

       // Axis V - Position Set point  according to start request
       IF #sFixtureUnloading.oAxisV_StartReq THEN
           #oAxisV_PosSetPoint := #sFixtureUnloading.oAxisV_PosSetPoint;
       ELSIF #sFixtureLoading.oAxisV_StartReq THEN
           #oAxisV_PosSetPoint := #sFixtureLoading.oAxisV_PosSetPoint;
       ELSIF #sFixtureBlowing.oAxisV_StartReq THEN
           #oAxisV_PosSetPoint := #sFixtureBlowing.oAxisV_PosSetPoint;
       ELSIF #sFixtureRelease.oAxisV_StartReq THEN
           #oAxisV_PosSetPoint := #sFixtureRelease.oAxisV_PosSetPoint;
       ELSIF #sFixtureV_Init.oAxisV_StartReq THEN
           #oAxisV_PosSetPoint := #sFixtureV_Init.oAxisV_PosSetPoint;
       ELSE
           #oAxisV_StartReq := FALSE;
       END_IF;

       // Axis W - Start Request
       #oAxisW_StartReq :=
       #sFixtureUnloading.oAxisW_StartReq
       OR #sFixtureLoading.oAxisW_StartReq
       OR #sFixtureBlowing.oAxisW_StartReq
       OR #sFixtureRelease.oAxisW_StartReq
       OR #sFixtureW_Init.iAxisW_StartReq;

       // Axis W - Position Set point  according to start request
       IF #sFixtureUnloading.oAxisW_StartReq THEN
           #oAxisW_PosSetPoint := #sFixtureUnloading.oAxisW_PosSetPoint;
       ELSIF #sFixtureLoading.oAxisW_StartReq THEN
           #oAxisW_PosSetPoint := #sFixtureLoading.oAxisW_PosSetPoint;
       ELSIF #sFixtureBlowing.oAxisW_StartReq THEN
           #oAxisW_PosSetPoint := #sFixtureBlowing.oAxisW_PosSetPoint;
       ELSIF #sFixtureRelease.oAxisW_StartReq THEN
           #oAxisW_PosSetPoint := #sFixtureRelease.oAxisW_PosSetPoint;
       ELSIF #sFixtureW_Init.iAxisW_StartReq THEN
           #oAxisW_PosSetPoint := #sFixtureW_Init.iAxisW_PosSetPoint;
       ELSE
           #oAxisW_StartReq := FALSE;
       END_IF;
   END_REGION


   REGION Gripper Command Request
       // Load Gripper
       #oLoadGripperOpenReq := #sFixtureLoading.oLoadGripperOpenReq;
       // Unload Gripper
       #oUnloadGripperCloseReq := #sFixtureUnloading.oUnloadGripperCloseReq;
   END_REGION

   REGION Fixture Command Request
       #oFixtureOpenReq := #sFixtureUnloading.oFixtureOpenReq
       OR #sFixtureLoading.oFixtureOpenReq
       OR #sFixtureBlowing.oFixtureOpenReq;

       #oFixtureCloseReq := #sFixtureLoading.oFixtureCloseReq;
   END_REGION

   REGION Blowing Command Request
       #oBlowingReq := #sFixtureBlowing.oBlowingReq;
   END_REGION

   REGION Message Waiting for Product
       "LBP_AlarmMsgs".UserA[03].A70UUxx[48] := #sFixtureMain.oNC_RID1;
   END_REGION
END_FUNCTION_BLOCK

FUNCTION_BLOCK "FB_FixtureUnloadLoad"   // FB65, SCL
{ S7_Optimized_Access := 'TRUE' }
// stored: MemoryReserve 100, SetENOAutomatically false
   VAR_INPUT
      iFixtureUnloadingRequest : Bool;
      iFixtureLoadingRequest : Bool;
      iFixtureBlowingRequest : Bool;
      iFixtureReleaseRequest : Bool;
      iFixtureV_InitRequest : Bool;
      iFixtureW_InitRequest : Bool;
      iWorkingModeFilling : Bool;
      iWorkingModeEmptying : Bool;
      iGripperReadyForUnloading : Bool;
      iGripperReadyForLoading : Bool;
      iGripperReadyForBlowing : Bool;
      iGripperReadyForRelease : Bool;
      iGripperReadyForV_Init : Bool;
      iGripperReadyForW_Init : Bool;
      iFixtureReadyForUnloading : Bool;
      iFixtureReadyForLoading : Bool;
      iFixtureReadyForBlowing : Bool;
      iFixtureReadyForRelease : Bool;
      iFixtureReadyForV_Init : Bool;
      iFixtureReadyForW_Init : Bool;
      iAxisReadyForUnloading : Bool;
      iAxisReadyForLoading : Bool;
      iAxisReadyForBlowing : Bool;
      iAxisReadyForRelease : Bool;
      iAxisReadyForV_Init : Bool;
      iAxisReadyForW_Init : Bool;
      iAxisV_W_Available : Bool;
   END_VAR
   VAR_OUTPUT
      oAxisV_W_Reservation : Bool;
      oNC_RID1 : Bool;
      oNC_RID2 : Bool;
   END_VAR
   VAR_IN_OUT
      ioFixtureUnloadingSeq : "UDT_SequenceInterface";
      ioFixtureLoadingSeq : "UDT_SequenceInterface";
      ioFixtureBlowingSeq : "UDT_SequenceInterface";
      ioFixtureReleaseSeq : "UDT_SequenceInterface";
      ioFixtureV_InitSeq : "UDT_SequenceInterface";
      ioFixtureW_InitSeq : "UDT_SequenceInterface";
   END_VAR
   VAR
      sRT_FixtureUnloadingRequest : R_TRIG;
      sRT_FixtureLoadingRequest { S7_SetPoint := 'True'} : R_TRIG;
      sRT_FixtureBlowingRequest { S7_SetPoint := 'True'} : R_TRIG;
      sRT_FixtureReleaseRequest { S7_SetPoint := 'True'} : R_TRIG;
      sRT_FixtureV_InitRequest { S7_SetPoint := 'True'} : R_TRIG;
      sRT_FixtureW_InitRequest { S7_SetPoint := 'True'} : R_TRIG;
      sMemoUnloadingRequest { S7_SetPoint := 'True'} : Bool;
      sMemoLoadingRequest { S7_SetPoint := 'True'} : Bool;
      sMemoBlowingRequest { S7_SetPoint := 'True'} : Bool;
      sMemoReleaseRequest { S7_SetPoint := 'True'} : Bool;
      sMemoV_InitRequest : Bool;
      sMemoW_InitRequest : Bool;
      sTONUnloadingNotFinished : TON_TIME;
      sTONBlowingNotFinished { S7_SetPoint := 'True'} : TON_TIME;
      sTONLoadingNotFinished { S7_SetPoint := 'True'} : TON_TIME;
   END_VAR
BEGIN
   REGION Description header 
       //==================================================================================
       // POSALUX Swiss SA / (C) Copyright 2026
       //----------------------------------------------------------------------------------
       // Title: FB_FixtureUnloadLoadMain
       // Comment/Function: 
       // Author: Fabien WALDT
       // Engineering: TIA Portal v20
       //----------------------------------------------------------------------------------
       // Change log table:
       // Version  | Date     | Expert in charge | Changes applied
       // ---------|----------|------------------|-----------------------------------------
       // 00.00.01 | 20260122 | WFA              | First released version
       // =================================================================================
   END_REGION

   REGION Init
       IF "LBP_Chan1".A_Reset THEN
           #oAxisV_W_Reservation := FALSE;
           #oNC_RID1 := FALSE;
           #oNC_RID2 := FALSE;
           #ioFixtureUnloadingSeq.StartRequest := FALSE;
           #ioFixtureLoadingSeq.StartRequest := FALSE;
           #ioFixtureBlowingSeq.StartRequest := FALSE;
           #ioFixtureReleaseSeq.StartRequest := FALSE;
           #ioFixtureV_InitSeq.StartRequest := FALSE;
           #ioFixtureW_InitSeq.StartRequest := FALSE;
           #sMemoUnloadingRequest := FALSE;
           #sMemoLoadingRequest := FALSE;
           #sMemoBlowingRequest := FALSE;
           #sMemoReleaseRequest := FALSE;
       END_IF;
   END_REGION

   REGION Fixture Unload Request
       #sRT_FixtureUnloadingRequest(CLK := #iFixtureUnloadingRequest        // M Code
                                    AND NOT #iWorkingModeFilling            // Not Mode Filling (No Part on Fixture)
                                    AND NOT (#iWorkingModeEmptying AND "DB_PartManagement".sPosition.sFixtureEmpty AND "DB_PartManagement".sPosition.sGripperEmpty)); // Not Gripper and Fixture Empty
       IF #sRT_FixtureUnloadingRequest.Q THEN
           #oNC_RID2 := TRUE;
           #sMemoUnloadingRequest := TRUE;
           "DB_LoaderFixtureMain".sBlowingNotFinished := FALSE;
           "DB_LoaderFixtureMain".sLoadingNotFinished := FALSE;
           "DB_LoaderFixtureMain".sUnloadingNotFinished := FALSE;
       END_IF;

       IF #sMemoUnloadingRequest
           AND #iGripperReadyForUnloading
           AND #iFixtureReadyForUnloading
           AND #iAxisReadyForUnloading
           AND NOT #iWorkingModeFilling
           AND NOT (#iWorkingModeEmptying AND "DB_PartManagement".sPosition.sFixtureEmpty AND "DB_PartManagement".sPosition.sGripperEmpty) THEN
           #oAxisV_W_Reservation := TRUE;
           #ioFixtureUnloadingSeq.StartRequest := TRUE;
       END_IF;

       #sTONUnloadingNotFinished(IN := "DB_LoaderFixtureMain".sUnloadingNotFinished,
                                 PT := T#100ms);

       IF #ioFixtureUnloadingSeq.JobDone
           OR "DB_LoaderFixtureMain".sUnloadingNotFinished THEN
           #ioFixtureUnloadingSeq.StartRequest := FALSE;
           #sMemoUnloadingRequest := FALSE;
       END_IF;

       IF #ioFixtureUnloadingSeq.JobDone
           OR #sTONUnloadingNotFinished.Q THEN
           #oNC_RID2 := FALSE;
       END_IF;
   END_REGION

   REGION Fixture Load Request
       #sRT_FixtureLoadingRequest(CLK := #iFixtureLoadingRequest
                                  AND NOT (#iWorkingModeEmptying AND NOT "DB_PartManagement".sPosition.sGripper.Undrilled.Presence.Part));
       IF #sRT_FixtureLoadingRequest.Q THEN
           #oNC_RID2 := TRUE;
           #sMemoLoadingRequest := TRUE;
           "DB_LoaderFixtureMain".sBlowingNotFinished := FALSE;
           "DB_LoaderFixtureMain".sLoadingNotFinished := FALSE;
           "DB_LoaderFixtureMain".sUnloadingNotFinished := FALSE;
       END_IF;

       IF #sMemoLoadingRequest
           AND #iGripperReadyForLoading
           AND #iFixtureReadyForLoading
           AND #iAxisReadyForLoading THEN
           #oAxisV_W_Reservation := TRUE;
           #ioFixtureLoadingSeq.StartRequest := TRUE;
       END_IF;

       #sTONLoadingNotFinished(IN := "DB_LoaderFixtureMain".sLoadingNotFinished,
                                 PT := T#100ms);

       IF #ioFixtureLoadingSeq.JobDone
           OR "DB_LoaderFixtureMain".sLoadingNotFinished THEN
           #ioFixtureLoadingSeq.StartRequest := FALSE;
           #sMemoLoadingRequest := FALSE;
       END_IF;

       IF #ioFixtureLoadingSeq.JobDone
           OR #sTONLoadingNotFinished.Q THEN
           #oNC_RID2 := FALSE;
       END_IF;
   END_REGION

   REGION Fixture Blowing Request
       #sRT_FixtureBlowingRequest(CLK := #iFixtureBlowingRequest
                                  AND NOT (#iWorkingModeEmptying AND NOT "DB_PartManagement".sPosition.sGripper.Undrilled.Presence.Part));
       IF #sRT_FixtureBlowingRequest.Q THEN
           #oNC_RID2 := TRUE;
           #sMemoBlowingRequest := TRUE;
           "DB_LoaderFixtureMain".sBlowingNotFinished := FALSE;
           "DB_LoaderFixtureMain".sLoadingNotFinished := FALSE;
           "DB_LoaderFixtureMain".sUnloadingNotFinished := FALSE;
       END_IF;

       IF #sMemoBlowingRequest
           AND #iGripperReadyForBlowing
           AND #iFixtureReadyForBlowing
           AND #iAxisReadyForBlowing THEN
           #oAxisV_W_Reservation := TRUE;
           #ioFixtureBlowingSeq.StartRequest := TRUE;
       END_IF;

       #sTONBlowingNotFinished(IN := "DB_LoaderFixtureMain".sBlowingNotFinished,
                               PT := T#100ms);

       IF #ioFixtureBlowingSeq.JobDone
       OR "DB_LoaderFixtureMain".sBlowingNotFinished THEN
           #ioFixtureBlowingSeq.StartRequest := FALSE;
           #sMemoBlowingRequest := FALSE;
       END_IF;

       IF #ioFixtureBlowingSeq.JobDone
           OR #sTONBlowingNotFinished.Q THEN
           #oNC_RID2 := FALSE;
       END_IF;
   END_REGION

   REGION Fixture Release Request
       #sRT_FixtureReleaseRequest(CLK := #iFixtureReleaseRequest
                                  OR #ioFixtureLoadingSeq.JobDone
                                  OR (#ioFixtureUnloadingSeq.JobDone AND (#iWorkingModeEmptying AND NOT "DB_PartManagement".sPosition.sGripper.Undrilled.Presence.Part)));
       // IF #sRT_FixtureReleaseRequest.Q THEN
       //     #oNC_RID2 := TRUE;
       //     #sMemoReleaseRequest := TRUE;
       // END_IF;

       IF (#sMemoReleaseRequest OR #ioFixtureLoadingSeq.JobDone
           OR (#ioFixtureUnloadingSeq.JobDone
           AND (#iWorkingModeEmptying AND NOT "DB_PartManagement".sPosition.sGripper.Undrilled.Presence.Part)))
           AND #iGripperReadyForRelease
           AND #iFixtureReadyForRelease
           AND #iAxisReadyForRelease THEN
           #oAxisV_W_Reservation := TRUE;
           #ioFixtureReleaseSeq.StartRequest := TRUE;
       END_IF;

       IF #ioFixtureReleaseSeq.JobDone
       OR "DB_LoaderFixtureMain".sReleaseNotFinished THEN
           #ioFixtureReleaseSeq.StartRequest := FALSE;
           #sMemoReleaseRequest := FALSE;
           #oNC_RID2 := FALSE;
           #oAxisV_W_Reservation := FALSE;
       END_IF;
   END_REGION

   REGION V Init Request
       #sRT_FixtureV_InitRequest(CLK := #iFixtureV_InitRequest);
       IF #sRT_FixtureV_InitRequest.Q THEN
           #oNC_RID1 := TRUE;
           #sMemoV_InitRequest := TRUE;
       END_IF;

       IF #sMemoV_InitRequest
           AND #iGripperReadyForV_Init
           AND #iFixtureReadyForV_Init
           AND #iAxisReadyForV_Init THEN
               #oAxisV_W_Reservation := TRUE;
               #ioFixtureV_InitSeq.StartRequest := TRUE;
       END_IF;

       IF #ioFixtureV_InitSeq.JobDone
       OR "DB_LoaderFixtureMain".sV_InitNotFinished THEN
           #ioFixtureV_InitSeq.StartRequest := FALSE;
           #sMemoV_InitRequest := FALSE;
           #oNC_RID1 := FALSE;
           #oAxisV_W_Reservation := FALSE;
       END_IF;
   END_REGION

   REGION W Init Request
       #sRT_FixtureW_InitRequest(CLK := #iFixtureW_InitRequest);
       IF #sRT_FixtureW_InitRequest.Q THEN
           #oNC_RID1 := TRUE;
           #sMemoW_InitRequest := TRUE;
       END_IF;

       IF #sMemoW_InitRequest
           AND #iGripperReadyForW_Init
           AND #iFixtureReadyForW_Init
           AND #iAxisReadyForW_Init THEN
           #oAxisV_W_Reservation := TRUE;
           #ioFixtureW_InitSeq.StartRequest := TRUE;
       END_IF;

       IF #ioFixtureW_InitSeq.JobDone
       OR "DB_LoaderFixtureMain".sW_InitNotFinished THEN
           #ioFixtureW_InitSeq.StartRequest := FALSE;
           #sMemoW_InitRequest := FALSE;
           #oNC_RID1 := FALSE;
           #oAxisV_W_Reservation := FALSE;
       END_IF;
   END_REGION
END_FUNCTION_BLOCK

FUNCTION_BLOCK "FB_FixtureUnloading"   // FB66, SCL
{ S7_Optimized_Access := 'TRUE' }
// stored: AutoNumber false, MemoryReserve 100, SetENOAutomatically false
   VAR_INPUT
      iStartSeqCond : Bool;   // Start Sequence Conditions
      iJobReq : Bool;   // Job Request - From Main
      iFixtureOpened : Bool;
      iUnloadGripperClosed : Bool;
      iAxisV_FixtUnloadPos : Bool;
      iAxisV_FixtUnloadPosSetPoint : LReal;
      iAxisW_FixtSafePos : Bool;
      iAxisW_FixtSafePosSetPoint : LReal;
      iAxisW_FixtUnloadPos : Bool;
      iAxisW_FixtUnloadPosSetPoint : LReal;
      iAxisV_Moving : Bool;   // Shuttle is moving
      iAxisV_InPos : Bool;
      iAxisW_Moving { ExternalAccessible := 'False'; ExternalVisible := 'False'; ExternalWritable := 'False'} : Bool;   // Shuttle is moving
      iAxisW_InPos : Bool;
      iPLC_DateAndTime : DTL;
      iStepPause : Bool;
   END_VAR
   VAR_OUTPUT
      oFixtureOpenReq : Bool;
      oUnloadGripperCloseReq : Bool;
      oVacuumStopReq : Bool;
      oAxisV_StartReq : Bool;
      oAxisV_PosSetPoint : Real;
      oAxisW_StartReq : Bool;
      oAxisW_PosSetPoint : Real;
   END_VAR
   VAR
      sCurrent_Step_NB : Int;   // Active Step Number
      sCheck_Step_Condition : Bool;
      sOneStepForward : Bool;
      sRTOneStepForward : R_TRIG;
      sOneStepMode { S7_SetPoint := 'True'} : Bool;
      sStepForward : Bool;
      sInterface : "UDT_SequenceInterface";
      sFixtureOpenReq { S7_SetPoint := 'True'} : Bool;
      sUnloadGripperCloseReq : Bool;
      sVacuumStopReq : Bool;
      sAxisV_StartReq : Bool;
      sAxisV_PosSetPoint : Real;
      sAxisW_StartReq : Bool;
      sAxisW_PosSetPoint : Real;
      sTimerFixtureOpened : TON_TIME;
      sTimerUnloadGripperClosed { S7_SetPoint := 'True'} : TON_TIME;
      sHistory : Struct
         Activation : Bool;
         Steps : Array[0..99] of Int;
         Date_Time : Array[0..99] of DTL;
      END_STRUCT;
      StepText : "FB_GetTextErrorCode";
   END_VAR
   VAR_TEMP
      tIndex : Int;   // Index
   END_VAR
   VAR CONSTANT
      S00_INIT : Int := 0;
      S10_CHECK_FIXTURE_UNLOAD_OPTION : Int := 10;
      S20_AXIS_W_TO_FIXTURE_SAFE_POS_START_REQ : Int := 20;
      S30_AXIS_W_TO_FIXTURE_SAFE_POS_REACHED : Int := 30;
      S40_AXIS_V_TO_FIXTURE_UNLOAD_POS_START_REQ : Int := 40;
      S50_AXIS_V_TO_FIXTURE_UNLOAD_POS_REACHED : Int := 50;
      S60_OPEN_FIXTURE : Int := 60;
      S70_AXIS_W_TO_FIXTURE_UNLOAD_POS_START_REQ : Int := 70;
      S80_AXIS_W_TO_FIXTURE_UNLOAD_POS_REACHED : Int := 80;
      S90_CLOSE_UNLOAD_GRIPPER : Int := 90;
      S95_VACUUM_STOP : Int := 95;
      S100_AXIS_W_TO_FIXTURE_SAFE_POS_START_REQ : Int := 100;
      S110_AXIS_W_TO_FIXTURE_SAFE_POS_REACHED : Int := 110;
      S195_JOB_DONE : Int := 195;
   END_VAR
   // StepText.sCode_error[0].ErrorCode := 0;
   // StepText.sCode_error[1].ErrorCode := 10;
   // StepText.sCode_error[2].ErrorCode := 20;
   // StepText.sCode_error[3].ErrorCode := 30;
   // StepText.sCode_error[4].ErrorCode := 40;
   // StepText.sCode_error[5].ErrorCode := 50;
   // StepText.sCode_error[6].ErrorCode := 60;
   // StepText.sCode_error[7].ErrorCode := 70;
   // StepText.sCode_error[8].ErrorCode := 80;
   // StepText.sCode_error[9].ErrorCode := 90;
   // StepText.sCode_error[10].ErrorCode := 95;
BEGIN
   REGION Description header 
       //==================================================================================
       // POSALUX Swiss SA / (C) Copyright 2026
       //----------------------------------------------------------------------------------
       // Title: FB_FixtureUnloading
       // Comment/Function: 
       // Author: Fabien WALDT
       // Engineering: TIA Portal v20
       //----------------------------------------------------------------------------------
       // Change log table:
       // Version  | Date     | Expert in charge | Changes applied
       // ---------|----------|------------------|-----------------------------------------
       // 00.00.01 | 20260122 | WFA              | First released version
       // =================================================================================
   END_REGION

   REGION Define condition to start
       IF #iStartSeqCond THEN
           #sInterface.SequenceReleased := TRUE;
       ELSE
           // Standard sequencer controls
           #sInterface.SequenceReleased := FALSE;
           #sCurrent_Step_NB := #S00_INIT;
           #sInterface.SequenceRun := FALSE;
           #sInterface.JobDone := FALSE;
           #sCheck_Step_Condition := FALSE;

           // Dedicated sequencer controls
           #sAxisV_StartReq := FALSE;
           #sAxisV_PosSetPoint := 0.0;
           #sAxisW_StartReq := FALSE;
           #sAxisW_PosSetPoint := 0.0;
           #sFixtureOpenReq := FALSE;
           #sUnloadGripperCloseReq := FALSE;
           #sVacuumStopReq := FALSE;

           // Add specifics controls 
       END_IF;

       // Reset interface error
       IF #sInterface.Reset THEN
           #sInterface.Error := FALSE;
       END_IF;

       // Reset start when axis in position
       IF #iAxisV_InPos THEN
           #sAxisV_StartReq := FALSE;
       END_IF;
       IF #iAxisW_InPos THEN
           #sAxisW_StartReq := FALSE;
       END_IF;

       // One step forward
       #sRTOneStepForward.CLK := #sOneStepForward;
       #sRTOneStepForward();
       #sStepForward := (NOT #sOneStepMode OR (#sOneStepMode AND #sRTOneStepForward.Q)) AND NOT #iStepPause;
       #sOneStepForward := FALSE;

       // Action only true in dedicated steps
       #sFixtureOpenReq := FALSE;
       #sUnloadGripperCloseReq := FALSE;
       #sVacuumStopReq := FALSE;

       // Step Timer
       #sTimerFixtureOpened(IN := #sCurrent_Step_NB = 60 AND #iFixtureOpened,
                          PT := T#200ms);

       #sTimerUnloadGripperClosed(IN := #sCurrent_Step_NB = 90 AND #iUnloadGripperClosed,
                                  PT := T#500ms);
   END_REGION

   REGION Sequence Function
       CASE #sCurrent_Step_NB OF
           #S00_INIT:
               REGION S00 INIT
                   #sCheck_Step_Condition := TRUE;
               END_REGION
           #S10_CHECK_FIXTURE_UNLOAD_OPTION:
               REGION S10_CHECK_FIXTURE_UNLOAD_OPTION
                   #sCheck_Step_Condition := TRUE;
               END_REGION
           #S20_AXIS_W_TO_FIXTURE_SAFE_POS_START_REQ:
               REGION S20_AXIS_W_TO_FIXTURE_SAFE_POS_START_REQ
                   #sAxisW_StartReq := NOT #iAxisW_FixtSafePos;
                   #sAxisW_PosSetPoint := LREAL_TO_REAL(#iAxisW_FixtSafePosSetPoint);
                   #sCheck_Step_Condition := TRUE;
               END_REGION
           #S30_AXIS_W_TO_FIXTURE_SAFE_POS_REACHED:
               REGION S30_AXIS_W_TO_FIXTURE_SAFE_POS_REACHED
                   #sCheck_Step_Condition := TRUE;
               END_REGION
           #S40_AXIS_V_TO_FIXTURE_UNLOAD_POS_START_REQ:
               REGION S40_AXIS_V_TO_FIXTURE_UNLOAD_POS_START_REQ
                   #sAxisV_StartReq := NOT #iAxisV_FixtUnloadPos;
                   #sAxisV_PosSetPoint := LREAL_TO_REAL(#iAxisV_FixtUnloadPosSetPoint);
                   #sCheck_Step_Condition := TRUE;
               END_REGION
           #S50_AXIS_V_TO_FIXTURE_UNLOAD_POS_REACHED:
               REGION S50_AXIS_V_TO_FIXTURE_UNLOAD_POS_REACHED
                   #sCheck_Step_Condition := TRUE;
               END_REGION
           #S60_OPEN_FIXTURE:
               REGION S60_OPEN_FIXTURE
                   #sFixtureOpenReq := TRUE;
                   IF #sTimerFixtureOpened.Q THEN
                       #sCheck_Step_Condition := TRUE;
                   END_IF;
               END_REGION
           #S70_AXIS_W_TO_FIXTURE_UNLOAD_POS_START_REQ:
               REGION S70_AXIS_W_TO_FIXTURE_UNLOAD_POS_START_REQ
                   #sAxisW_StartReq := NOT #iAxisW_FixtUnloadPos;
                   #sAxisW_PosSetPoint := LREAL_TO_REAL(#iAxisW_FixtUnloadPosSetPoint);
                   #sCheck_Step_Condition := TRUE;
               END_REGION
           #S80_AXIS_W_TO_FIXTURE_UNLOAD_POS_REACHED:
               REGION S80_AXIS_W_TO_FIXTURE_UNLOAD_POS_REACHED
                   #sCheck_Step_Condition := TRUE;
               END_REGION
           #S90_CLOSE_UNLOAD_GRIPPER:
               REGION S90_CLOSE_UNLOAD_GRIPPER
                   #sUnloadGripperCloseReq := TRUE;
                   IF #sTimerUnloadGripperClosed.Q THEN
                       #sCheck_Step_Condition := TRUE;
                   END_IF;
               END_REGION
           #S95_VACUUM_STOP:
               REGION S95_VACUUM_STOP
                   #sVacuumStopReq := TRUE;
                   #sCheck_Step_Condition := TRUE;
               END_REGION
           #S100_AXIS_W_TO_FIXTURE_SAFE_POS_START_REQ:
               REGION S100_AXIS_W_TO_FIXTURE_SAFE_POS_START_REQ
                   #sAxisW_StartReq := NOT #iAxisW_FixtSafePos;
                   #sAxisW_PosSetPoint := LREAL_TO_REAL(#iAxisW_FixtSafePosSetPoint);
                   #sCheck_Step_Condition := TRUE;
               END_REGION
           #S110_AXIS_W_TO_FIXTURE_SAFE_POS_REACHED:
               REGION S110_AXIS_W_TO_FIXTURE_SAFE_POS_REACHED
                   #sCheck_Step_Condition := TRUE;
               END_REGION
           #S195_JOB_DONE:
               REGION S195_JOB_DONE
                   #sInterface.JobDone := TRUE;
                   #sCheck_Step_Condition := TRUE;
               END_REGION
           ELSE:
               #sInterface.Error := TRUE;
       END_CASE;
   END_REGION

   REGION Sequence Next Step Condition
       IF #sCheck_Step_Condition THEN
           CASE #sCurrent_Step_NB OF
               #S00_INIT:
                   REGION S00_INIT
                       IF #sInterface.SequenceReleased AND #iJobReq THEN
                           #sCurrent_Step_NB := #S10_CHECK_FIXTURE_UNLOAD_OPTION;
                           #sInterface.SequenceRun := TRUE;
                           #sCheck_Step_Condition := FALSE;
                       ELSE
                           #sInterface.SequenceRun := FALSE;
                       END_IF;
                   END_REGION
               #S10_CHECK_FIXTURE_UNLOAD_OPTION:
                   REGION S10_CHECK_FIXTURE_UNLOAD_OPTION
                       IF #sInterface.SequenceReleased AND #sStepForward AND NOT "DB_LoaderOptions".Fixture.UnloadingDisabled  THEN
                           #sCurrent_Step_NB := #S20_AXIS_W_TO_FIXTURE_SAFE_POS_START_REQ;
                           #sCheck_Step_Condition := FALSE;
                       ELSIF #sInterface.SequenceReleased AND #sStepForward AND "DB_LoaderOptions".Fixture.UnloadingDisabled THEN
                           #sCurrent_Step_NB := #S195_JOB_DONE;
                           #sCheck_Step_Condition := FALSE;
                       END_IF;
                   END_REGION
               #S20_AXIS_W_TO_FIXTURE_SAFE_POS_START_REQ:
                   REGION S20_AXIS_W_TO_FIXTURE_SAFE_POS_START_REQ
                       IF #sInterface.SequenceReleased AND #sStepForward AND (#iAxisW_Moving OR #iAxisW_FixtSafePos) THEN
                           #sCurrent_Step_NB := #S30_AXIS_W_TO_FIXTURE_SAFE_POS_REACHED;
                           #sCheck_Step_Condition := FALSE;
                       END_IF;
                   END_REGION
               #S30_AXIS_W_TO_FIXTURE_SAFE_POS_REACHED:
                   REGION S30_AXIS_W_TO_FIXTURE_SAFE_POS_REACHED
                       IF #sInterface.SequenceReleased AND #sStepForward AND NOT #sAxisW_StartReq AND #iAxisW_FixtSafePos THEN
                           #sCurrent_Step_NB := #S40_AXIS_V_TO_FIXTURE_UNLOAD_POS_START_REQ;
                           #sCheck_Step_Condition := FALSE;
                       END_IF;
                   END_REGION
               #S40_AXIS_V_TO_FIXTURE_UNLOAD_POS_START_REQ:
                   REGION S40_AXIS_V_TO_FIXTURE_UNLOAD_POS_START_REQ
                       IF #sInterface.SequenceReleased AND #sStepForward AND (#iAxisV_Moving OR #iAxisV_FixtUnloadPos) THEN
                           #sCurrent_Step_NB := #S50_AXIS_V_TO_FIXTURE_UNLOAD_POS_REACHED;
                           #sCheck_Step_Condition := FALSE;
                       END_IF;
                   END_REGION
               #S50_AXIS_V_TO_FIXTURE_UNLOAD_POS_REACHED:
                   REGION S50_AXIS_V_TO_FIXTURE_UNLOAD_POS_REACHED
                       IF #sInterface.SequenceReleased AND #sStepForward AND NOT #sAxisV_StartReq AND #iAxisV_FixtUnloadPos THEN
                           #sCurrent_Step_NB := #S60_OPEN_FIXTURE;
                           #sCheck_Step_Condition := FALSE;
                       END_IF;
                   END_REGION
               #S60_OPEN_FIXTURE:
                   REGION S60_OPEN_FIXTURE
                       IF #sInterface.SequenceReleased AND #sStepForward AND #iFixtureOpened THEN
                           #sCurrent_Step_NB := #S70_AXIS_W_TO_FIXTURE_UNLOAD_POS_START_REQ;
                           #sCheck_Step_Condition := FALSE;
                       END_IF;
                   END_REGION
               #S70_AXIS_W_TO_FIXTURE_UNLOAD_POS_START_REQ:
                   REGION S70_AXIS_W_TO_FIXTURE_UNLOAD_POS_START_REQ
                       IF #sInterface.SequenceReleased AND #sStepForward AND (#iAxisW_Moving OR #iAxisW_FixtUnloadPos) THEN
                           #sCurrent_Step_NB := #S80_AXIS_W_TO_FIXTURE_UNLOAD_POS_REACHED;
                           #sCheck_Step_Condition := FALSE;
                       END_IF;
                   END_REGION
               #S80_AXIS_W_TO_FIXTURE_UNLOAD_POS_REACHED:
                   REGION S80_AXIS_W_TO_FIXTURE_UNLOAD_POS_REACHED
                       IF #sInterface.SequenceReleased AND #sStepForward AND NOT #sAxisW_StartReq AND #iAxisW_FixtUnloadPos THEN
                           #sCurrent_Step_NB := #S90_CLOSE_UNLOAD_GRIPPER;
                           #sCheck_Step_Condition := FALSE;
                       END_IF;
                   END_REGION
               #S90_CLOSE_UNLOAD_GRIPPER:
                   REGION S90_CLOSE_UNLOAD_GRIPPER
                       IF #sInterface.SequenceReleased AND #sStepForward AND #iUnloadGripperClosed THEN
                           #sCurrent_Step_NB := #S95_VACUUM_STOP;
                           #sCheck_Step_Condition := FALSE;
                       END_IF;
                   END_REGION
               #S95_VACUUM_STOP:
                   REGION S95_VACUUM_STOP
                       IF #sInterface.SequenceReleased AND #sStepForward AND TRUE THEN
                           #sCurrent_Step_NB := #S100_AXIS_W_TO_FIXTURE_SAFE_POS_START_REQ;
                           #sCheck_Step_Condition := FALSE;
                       END_IF;
                   END_REGION
               #S100_AXIS_W_TO_FIXTURE_SAFE_POS_START_REQ:
                   REGION S100_AXIS_W_TO_FIXTURE_SAFE_POS_START_REQ
                       IF #sInterface.SequenceReleased AND #sStepForward AND (#iAxisW_Moving OR #iAxisW_FixtSafePos) THEN
                           #sCurrent_Step_NB := #S110_AXIS_W_TO_FIXTURE_SAFE_POS_REACHED;
                           #sCheck_Step_Condition := FALSE;
                       END_IF;
                   END_REGION
               #S110_AXIS_W_TO_FIXTURE_SAFE_POS_REACHED:
                   REGION S110_AXIS_W_TO_FIXTURE_SAFE_POS_REACHED
                       IF #sInterface.SequenceReleased AND #sStepForward AND NOT #sAxisW_StartReq AND #iAxisW_FixtSafePos THEN
                           #sCurrent_Step_NB := #S195_JOB_DONE;
                           #sCheck_Step_Condition := FALSE;
                       END_IF;
                   END_REGION
               #S195_JOB_DONE:
                   REGION S195_JOB_DONE
                       IF NOT #iJobReq THEN
                           #sCurrent_Step_NB := #S00_INIT;
                           #sCheck_Step_Condition := FALSE;
                           #sInterface.JobDone := FALSE;
                       END_IF;
                   END_REGION
               ELSE
                   #sInterface.Error := TRUE;
           END_CASE;
       END_IF;
   END_REGION

   REGION Outputs Update
       #oAxisV_StartReq := #sAxisV_StartReq;
       #oAxisV_PosSetPoint := #sAxisV_PosSetPoint;
       #oAxisW_StartReq := #sAxisW_StartReq;
       #oAxisW_PosSetPoint := #sAxisW_PosSetPoint;
       #oFixtureOpenReq := #sFixtureOpenReq;
       #oUnloadGripperCloseReq := #sUnloadGripperCloseReq;
       #oVacuumStopReq := #sVacuumStopReq;
   END_REGION

   REGION Steps - Date and Time History
       IF #sHistory.Activation THEN
           IF #sHistory.Steps[0] <> #sCurrent_Step_NB THEN
               FOR #tIndex := 98 TO 0 BY -1 DO
                   #sHistory.Steps[#tIndex + 1] := #sHistory.Steps[#tIndex];
                   #sHistory.Date_Time[#tIndex + 1] := #sHistory.Date_Time[#tIndex];
               END_FOR;
               #sHistory.Steps[0] := #sCurrent_Step_NB;
               #sHistory.Date_Time[0] := #iPLC_DateAndTime;
           END_IF;
       END_IF;
   END_REGION

   REGION Steps Text
       #StepText(iErrorCode := #sCurrent_Step_NB,
                 oErrorText => #StepText.oErrorText);
   END_REGION
END_FUNCTION_BLOCK

FUNCTION_BLOCK "FB_FixtureLoading"   // FB67, SCL
{ S7_Optimized_Access := 'TRUE' }
// stored: AutoNumber false, MemoryReserve 100, SetENOAutomatically false
   VAR_INPUT
      iStartSeqCond : Bool;   // Start Sequence Conditions
      iJobReq : Bool;   // Job Request - From Main
      iFixtureOpened : Bool;
      iFixtureClosed : Bool;
      iLoadGripperOpened : Bool;
      iAxisV_FixtLoadPos : Bool;
      iAxisV_FixtLoadPosSetPoint : LReal;
      iAxisW_FixtSafePos : Bool;
      iAxisW_FixtSafePosSetPoint : LReal;
      iAxisW_FixtLoadPos : Bool;
      iAxisW_FixtLoadPosSetPoint : LReal;
      iAxisW_FixtApproachPos : Bool;
      iAxisW_FixtApproachPosSetPoint : LReal;
      iAxisV_Moving : Bool;   // Shuttle is moving
      iAxisV_InPos : Bool;
      iAxisW_Moving { ExternalAccessible := 'False'; ExternalVisible := 'False'; ExternalWritable := 'False'} : Bool;   // Shuttle is moving
      iAxisW_InPos : Bool;
      iPLC_DateAndTime : DTL;
      iStepPause : Bool;
   END_VAR
   VAR_OUTPUT
      oFixtureOpenReq : Bool;
      oFixtureCloseReq : Bool;
      oLoadGripperOpenReq : Bool;
      oVacuumStartReq : Bool;
      oAxisV_StartReq : Bool;
      oAxisV_PosSetPoint : Real;
      oAxisW_StartReq : Bool;
      oAxisW_PosSetPoint : Real;
   END_VAR
   VAR
      sCurrent_Step_NB : Int;   // Active Step Number
      sCheck_Step_Condition : Bool;
      sOneStepForward : Bool;
      sRTOneStepForward : R_TRIG;
      sOneStepMode { S7_SetPoint := 'True'} : Bool;
      sStepForward : Bool;
      sInterface : "UDT_SequenceInterface";
      sFixtureOpenReq { S7_SetPoint := 'True'} : Bool;
      sFixtureCloseReq : Bool;
      sLoadGripperOpenReq : Bool;
      sVacuumStartReq : Bool;
      sAxisV_StartReq : Bool;
      sAxisV_PosSetPoint : Real;
      sAxisW_StartReq : Bool;
      sAxisW_PosSetPoint : Real;
      sTimerFixtureOpened : TON_TIME;
      sTimerFixtureClosed { S7_SetPoint := 'True'} : TON_TIME;
      sTimerLoadGripperOpened { S7_SetPoint := 'True'} : TON_TIME;
      sTimerAfterApproach { S7_SetPoint := 'True'} : TON_TIME;
      sHistory : Struct
         Activation : Bool;
         Steps : Array[0..99] of Int;
         Date_Time : Array[0..99] of DTL;
      END_STRUCT;
      StepText : "FB_GetTextErrorCode";
   END_VAR
   VAR_TEMP
      tIndex : Int;   // Index
   END_VAR
   VAR CONSTANT
      S00_INIT : Int := 0;
      S10_CHECK_FIXTURE_LOAD_OPTION : Int := 10;
      S20_AXIS_W_TO_FIXTURE_SAFE_POS_START_REQ : Int := 20;
      S30_AXIS_W_TO_FIXTURE_SAFE_POS_REACHED : Int := 30;
      S40_AXIS_V_TO_FIXTURE_LOAD_POS_START_REQ : Int := 40;
      S50_AXIS_V_TO_FIXTURE_LOAD_POS_REACHED : Int := 50;
      S60_OPEN_FIXTURE : Int := 60;
      S70_AXIS_W_TO_FIXTURE_APPROACH_POS_START_REQ : Int := 70;
      S75_AXIS_W_TO_FIXTURE_APPROACH_POS_REACHED : Int := 75;
      S80_AXIS_W_TO_FIXTURE_LOAD_POS_START_REQ : Int := 80;
      S85_AXIS_W_TO_FIXTURE_LOAD_POS_REACHED : Int := 85;
      S90_OPEN_LOAD_GRIPPER : Int := 90;
      S95_VACUUM_START : Int := 95;
      S100_AXIS_W_TO_FIXTURE_SAFE_POS_START_REQ : Int := 100;
      S110_AXIS_W_TO_FIXTURE_SAFE_POS_REACHED : Int := 110;
      S120_CLOSE_FIXTURE : Int := 120;
      S195_JOB_DONE : Int := 195;
   END_VAR
   // StepText.sCode_error[0].ErrorCode := 0;
   // StepText.sCode_error[1].ErrorCode := 10;
   // StepText.sCode_error[2].ErrorCode := 20;
   // StepText.sCode_error[3].ErrorCode := 30;
   // StepText.sCode_error[4].ErrorCode := 40;
   // StepText.sCode_error[5].ErrorCode := 50;
   // StepText.sCode_error[6].ErrorCode := 60;
   // StepText.sCode_error[7].ErrorCode := 70;
   // StepText.sCode_error[8].ErrorCode := 80;
   // StepText.sCode_error[9].ErrorCode := 90;
   // StepText.sCode_error[10].ErrorCode := 95;
BEGIN
   REGION Description header 
       //==================================================================================
       // POSALUX Swiss SA / (C) Copyright 2026
       //----------------------------------------------------------------------------------
       // Title: FB_FixtureLoading
       // Comment/Function: 
       // Author: Fabien WALDT
       // Engineering: TIA Portal v20
       //----------------------------------------------------------------------------------
       // Change log table:
       // Version  | Date     | Expert in charge | Changes applied
       // ---------|----------|------------------|-----------------------------------------
       // 00.00.01 | 20260122 | WFA              | First released version
       // =================================================================================
   END_REGION

   REGION Define condition to start
       IF #iStartSeqCond THEN
           #sInterface.SequenceReleased := TRUE;
       ELSE
           // Standard sequencer controls
           #sInterface.SequenceReleased := FALSE;
           #sCurrent_Step_NB := #S00_INIT;
           #sInterface.SequenceRun := FALSE;
           #sInterface.JobDone := FALSE;
           #sCheck_Step_Condition := FALSE;

           // Dedicated sequencer controls
           #sAxisV_StartReq := FALSE;
           #sAxisV_PosSetPoint := 0.0;
           #sAxisW_StartReq := FALSE;
           #sAxisW_PosSetPoint := 0.0;
           #sFixtureOpenReq := FALSE;
           #sLoadGripperOpenReq := FALSE;
           #sVacuumStartReq := FALSE;

           // Add specifics controls 
       END_IF;

       // Reset interface error
       IF #sInterface.Reset THEN
           #sInterface.Error := FALSE;
       END_IF;

       // Reset start when axis in position
       IF #iAxisV_InPos THEN
           #sAxisV_StartReq := FALSE;
       END_IF;
       IF #iAxisW_InPos THEN
           #sAxisW_StartReq := FALSE;
       END_IF;

       // One step forward
       #sRTOneStepForward.CLK := #sOneStepForward;
       #sRTOneStepForward();
       #sStepForward := (NOT #sOneStepMode OR (#sOneStepMode AND #sRTOneStepForward.Q)) AND NOT #iStepPause;
       #sOneStepForward := FALSE;

       // Action only true in dedicated steps
       #sFixtureOpenReq := FALSE;
       #sFixtureCloseReq := FALSE;
       #sLoadGripperOpenReq := FALSE;
       #sVacuumStartReq := FALSE;

       // Step Timer
       #sTimerFixtureOpened(IN := #sCurrent_Step_NB = 60 AND #iFixtureOpened,
                            PT := T#200ms);

       #sTimerFixtureClosed(IN := #sCurrent_Step_NB = 120 AND #iFixtureClosed,
                            PT := T#200ms);

